KUKA KRL program: EPS_2_25862_MH08_A_20251016035158.src

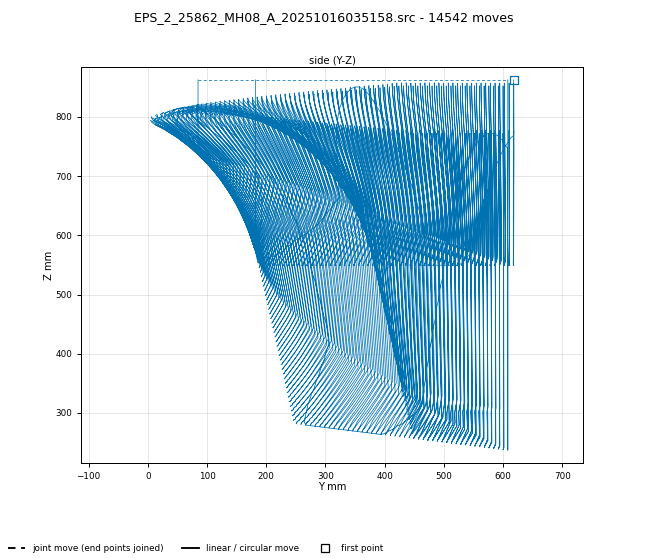
[picture p0: tool path of EPS_2_25862_MH08_A_20251016035158.src, 14542 of 14544 moves have a stored position in this frame; points joined in program order, loops and branches not executed]
&ACCESS RVP
&REL 4
&COMMENT QRS 19112012
&PARAM EDITMASK = *
DEF PART()
EXT BAS (BAS_COMMAND :IN,REAL :IN )
INT I
BAS (#INITMOV,0 )

;KUKA QRS Post kuka4.cps  Date:22-06-2017 !

File_ID=2888

QRS_PRE_INIT()

;Init var - Until changes are made in qrs_pre_init
Outlet_Square_prg=0
Inlet_1_Square_prg=0
Inlet_2_Square_prg=0
Inlet_3_Square_prg=0
Inlet_4_Square_prg=0
Inlet_5_Square_prg=0

Outlet_1={X 0.000, Y 425.000, Z 586.000, B 0.000, E1 0.000 }
Inlet_1={X 0.000, Y 425.000, Z 506.000, B 0.000, E1 105.000 }
Outlet_1_type=533
Inlet_1_type=533
;QRS#1=Sidecore dimensions
;QRS#2=525-21" Concrete
;QRS#3=525-21" Concrete
;QRS#4=
;QRS#5=
;QRS#6=
;QRS#7=
;QRS#8=
;QRS#9=S306-32
;QRS#10=S306-32
;QRS#11=
;QRS#12=
;QRS#13=
;QRS#14=
;QRS#15=
;QRS#16=1220x127x1219 4'
;QRS#17=EPS Height
;QRS#18=852,5
;QRS#19=*
;QRS#20= UPDATED VERSION 22-06-2017
;QRS#21=*
Outlet_Square=0250
Inlet_1_Square=0250
Inlet_2_Square=0
Inlet_3_Square=0
Inlet_4_Square=0
Inlet_5_Square=0
Mill_Square=1
Outlet_Square_Prg=263
Inlet_1_Square_prg=263

QRS_INIT()

$ADVANCE=5

; T1
PTP {E1 171.076,E2 171.076}
PTP {X 0,Y 617.86,A -85,B 0,C 180,E1 171.076,E2 171.076,E3 0,E4 0,E5 0,E6 0}
QRS_SPEED_INIT()
LIN {X 0,Y 617.86,Z 862.5,A -85,B 0,C 180,E1 171.076,E2 171.076,E3 0,E4 0,E5 0,E6 0} C_VEL
LIN {X 0,Y 617.86,Z 779.647,A -85,B 0,C 180,E1 171.076,E2 171.076} C_VEL
LIN {X 0,Y 617.86,Z 770.782,A -85,B 0,C 180,E1 171.076,E2 171.076} C_VEL
LIN {X 0,Y 617.855,Z 768.843,A -85,B 0,C 180,E1 171.216,E2 171.216} C_VEL
LIN {X 0,Y 617.946,Z 765.76,A -85,B 0,C 180,E1 172.353,E2 172.353} C_VEL
LIN {X 0,Y 617.789,Z 761.298,A -85,B 0,C 180,E1 173.748,E2 173.748} C_VEL
LIN {X 0,Y 617.856,Z 757.801,A -85,B 0,C 180,E1 174.678,E2 174.678} C_VEL
LIN {X 0,Y 618.003,Z 753.871,A -85,B 0,C 180,E1 175.607,E2 175.607} C_VEL
LIN {X 0,Y 617.888,Z 750.793,A -85,B 0,C 180,E1 176.301,E2 176.301} C_VEL
LIN {X 0,Y 617.795,Z 745.083,A -85,B 0,C 180,E1 177.458,E2 177.458} C_VEL
LIN {X 0,Y 617.882,Z 740.033,A -85,B 0,C 180,E1 178.384,E2 178.384} C_VEL
LIN {X 0,Y 617.968,Z 734.443,A -85,B 0,C 180,E1 179.308,E2 179.308} C_VEL
LIN {X 0,Y 617.83,Z 725.303,A -85,B 0,C 180,E1 180.695,E2 180.695} C_VEL
LIN {X 0,Y 617.888,Z 718.536,A -85,B 0,C 180,E1 181.619,E2 181.619} C_VEL
LIN {X 0,Y 617.931,Z 709.192,A -85,B 0,C 180,E1 182.776,E2 182.776} C_VEL
LIN {X 0,Y 617.867,Z 701.077,A -85,B 0,C 180,E1 183.702,E2 183.702} C_VEL
LIN {X 0,Y 617.921,Z 692.2,A -85,B 0,C 180,E1 184.628,E2 184.628} C_VEL
LIN {X 0,Y 617.95,Z 682.514,A -85,B 0,C 180,E1 185.556,E2 185.556} C_VEL
LIN {X 0,Y 617.899,Z 673.337,A -85,B 0,C 180,E1 186.37,E2 186.37} C_VEL
LIN {X 0,Y 617.909,Z 663.341,A -85,B 0,C 180,E1 187.184,E2 187.184} C_VEL
LIN {X 0,Y 617.892,Z 652.417,A -85,B 0,C 180,E1 188,E2 188} C_VEL
LIN {X 0,Y 617.911,Z 641.615,A -85,B 0,C 180,E1 188.738,E2 188.738} C_VEL
LIN {X 0,Y 617.886,Z 630.772,A -85,B 0,C 180,E1 189.418,E2 189.418} C_VEL
LIN {X 0,Y 617.869,Z 619.117,A -85,B 0,C 180,E1 190.08,E2 190.08} C_VEL
LIN {X 0,Y 617.915,Z 605.805,A -85,B 0,C 180,E1 190.752,E2 190.752} C_VEL
LIN {X 0,Y 617.872,Z 594.523,A -85,B 0,C 180,E1 191.268,E2 191.268} C_VEL
LIN {X 0,Y 617.78,Z 582.771,A -85,B 0,C 180,E1 191.749,E2 191.749} C_VEL
LIN {X 0,Y 617.848,Z 567.515,A -85,B 0,C 180,E1 192.274,E2 192.274} C_VEL
LIN {X 0,Y 617.736,Z 554.731,A -85,B 0,C 180,E1 192.655,E2 192.655} C_VEL
LIN {X 0,Y 617.593,Z 549.754,A -85,B 0,C 180,E1 192.788,E2 192.788} C_VEL
LIN {X 0,Y 617.736,Z 549.53,A -85,B 0,C 180,E1 192.822,E2 192.822} C_VEL
LIN {X 0,Y 618.063,Z 549.53,A -85,B 0,C 180,E1 192.963,E2 192.963} C_VEL
LIN {X 0,Y 617.964,Z 549.53,A -85,B 0,C 180,E1 195.199,E2 195.199} C_VEL
LIN {X 0,Y 617.909,Z 549.53,A -85,B 0,C 180,E1 200.051,E2 200.051} C_VEL
LIN {X 0,Y 617.429,Z 549.53,A -85,B 0,C 180,E1 202.55,E2 202.55} C_VEL
LIN {X 0,Y 617.883,Z 549.53,A -85,B 0,C 180,E1 205.058,E2 205.058} C_VEL
LIN {X 0,Y 617.396,Z 549.53,A -85,B 0,C 180,E1 207.661,E2 207.661} C_VEL
LIN {X 0,Y 617.869,Z 549.53,A -85,B 0,C 180,E1 210.28,E2 210.28} C_VEL
LIN {X 0,Y 617.313,Z 549.53,A -85,B 0,C 180,E1 213.028,E2 213.028} C_VEL
LIN {X 0,Y 617.774,Z 549.53,A -85,B 0,C 180,E1 215.802,E2 215.802} C_VEL
LIN {X 0,Y 617.556,Z 549.53,A -85,B 0,C 180,E1 218.097,E2 218.097} C_VEL
LIN {X 0,Y 617.539,Z 549.53,A -85,B 0,C 180,E1 218.724,E2 218.724} C_VEL
LIN {X 0,Y 617.773,Z 549.53,A -85,B 0,C 180,E1 221.734,E2 221.734} C_VEL
LIN {X 0,Y 617.845,Z 549.53,A -85,B 0,C 180,E1 225.096,E2 225.096} C_VEL
LIN {X 0,Y 617.433,Z 549.53,A -85,B 0,C 180,E1 228.311,E2 228.311} C_VEL
LIN {X 0,Y 617.775,Z 549.53,A -85,B 0,C 180,E1 231.294,E2 231.294} C_VEL
LIN {X 0,Y 617.721,Z 549.53,A -85,B 0,C 180,E1 235.803,E2 235.803} C_VEL
LIN {X 0,Y 617.906,Z 549.53,A -85,B 0,C 180,E1 237.008,E2 237.008} C_VEL
LIN {X 0,Y 618.058,Z 549.53,A -85,B 0,C 180,E1 240.653,E2 240.653} C_VEL
LIN {X 0,Y 617.765,Z 549.53,A -85,B 0,C 180,E1 240.802,E2 240.802} C_VEL
LIN {X 0,Y 617.424,Z 549.53,A -85,B 0,C 180,E1 240.866,E2 240.866} C_VEL
LIN {X 0,Y 617.177,Z 552.007,A -85,B 0,C 180,E1 240.934,E2 240.934} C_VEL
LIN {X 0,Y 617.712,Z 600.072,A -85,B 0,C 180,E1 241.593,E2 241.593} C_VEL
LIN {X 0,Y 617.671,Z 613,A -85,B 0,C 180,E1 241.802,E2 241.802} C_VEL
LIN {X 0,Y 617.749,Z 625.862,A -85,B 0,C 180,E1 242.077,E2 242.077} C_VEL
LIN {X 0,Y 617.69,Z 639.633,A -85,B 0,C 180,E1 242.435,E2 242.435} C_VEL
LIN {X 0,Y 617.845,Z 652.624,A -85,B 0,C 180,E1 242.849,E2 242.849} C_VEL
LIN {X 0,Y 617.868,Z 663.92,A -85,B 0,C 180,E1 243.255,E2 243.255} C_VEL
LIN {X 0,Y 617.757,Z 677.549,A -85,B 0,C 180,E1 243.815,E2 243.815} C_VEL
LIN {X 0,Y 617.88,Z 689.57,A -85,B 0,C 180,E1 244.383,E2 244.383} C_VEL
LIN {X 0,Y 617.885,Z 701.766,A -85,B 0,C 180,E1 245.021,E2 245.021} C_VEL
LIN {X 0,Y 617.847,Z 713.431,A -85,B 0,C 180,E1 245.696,E2 245.696} C_VEL
LIN {X 0,Y 617.909,Z 724.148,A -85,B 0,C 180,E1 246.381,E2 246.381} C_VEL
LIN {X 0,Y 617.926,Z 735.395,A -85,B 0,C 180,E1 247.169,E2 247.169} C_VEL
LIN {X 0,Y 617.917,Z 745.495,A -85,B 0,C 180,E1 247.938,E2 247.938} C_VEL
LIN {X 0,Y 617.886,Z 756.638,A -85,B 0,C 180,E1 248.868,E2 248.868} C_VEL
LIN {X 0,Y 617.923,Z 766.758,A -85,B 0,C 180,E1 249.796,E2 249.796} C_VEL
LIN {X 0,Y 617.933,Z 775.516,A -85,B 0,C 180,E1 250.667,E2 250.667} C_VEL
LIN {X 0,Y 617.881,Z 782.645,A -85,B 0,C 180,E1 251.423,E2 251.423} C_VEL
LIN {X 0,Y 617.901,Z 791.01,A -85,B 0,C 180,E1 252.391,E2 252.391} C_VEL
LIN {X 0,Y 617.982,Z 799.194,A -85,B 0,C 180,E1 253.428,E2 253.428} C_VEL
LIN {X 0,Y 617.836,Z 807.707,A -85,B 0,C 180,E1 254.61,E2 254.61} C_VEL
LIN {X 0,Y 617.888,Z 814.764,A -85,B 0,C 180,E1 255.696,E2 255.696} C_VEL
LIN {X 0,Y 617.959,Z 820.117,A -85,B 0,C 180,E1 256.59,E2 256.59} C_VEL
LIN {X 0,Y 617.783,Z 826.559,A -85,B 0,C 180,E1 257.772,E2 257.772} C_VEL
LIN {X 0,Y 617.807,Z 832.241,A -85,B 0,C 180,E1 258.952,E2 258.952} C_VEL
LIN {X 0,Y 617.978,Z 836.454,A -85,B 0,C 180,E1 259.948,E2 259.948} C_VEL
LIN {X 0,Y 617.803,Z 841.451,A -85,B 0,C 180,E1 261.248,E2 261.248} C_VEL
LIN {X 0,Y 617.803,Z 845.014,A -85,B 0,C 180,E1 262.349,E2 262.349} C_VEL
LIN {X 0,Y 617.954,Z 848.839,A -85,B 0,C 180,E1 263.748,E2 263.748} C_VEL
LIN {X 0,Y 617.79,Z 850.923,A -85,B 0,C 180,E1 264.675,E2 264.675} C_VEL
LIN {X 0,Y 617.737,Z 852.676,A -85,B 0,C 180,E1 265.603,E2 265.603} C_VEL
LIN {X 0,Y 617.832,Z 854.095,A -85,B 0,C 180,E1 266.53,E2 266.53} C_VEL
LIN {X 0,Y 617.873,Z 855.552,A -85,B 0,C 180,E1 267.919,E2 267.919} C_VEL
LIN {X 0,Y 617.747,Z 856.216,A -85,B 0,C 180,E1 268.843,E2 268.843} C_VEL
LIN {X 0,Y 617.993,Z 856.15,A -85,B 0,C 180,E1 271.154,E2 271.154} C_VEL
LIN {X 0,Y 617.755,Z 855.227,A -85,B 0,C 180,E1 272.542,E2 272.542} C_VEL
LIN {X 0,Y 617.805,Z 853.446,A -85,B 0,C 180,E1 273.931,E2 273.931} C_VEL
LIN {X 0,Y 617.985,Z 851.841,A -85,B 0,C 180,E1 274.857,E2 274.857} C_VEL
LIN {X 0,Y 617.799,Z 848.883,A -85,B 0,C 180,E1 276.252,E2 276.252} C_VEL
LIN {X 0,Y 617.849,Z 845.01,A -85,B 0,C 180,E1 277.649,E2 277.649} C_VEL
LIN {X 0,Y 617.932,Z 841.121,A -85,B 0,C 180,E1 278.829,E2 278.829} C_VEL
LIN {X 0,Y 617.775,Z 836.418,A -85,B 0,C 180,E1 280.074,E2 280.074} C_VEL
LIN {X 0,Y 617.826,Z 832.246,A -85,B 0,C 180,E1 281.046,E2 281.046} C_VEL
LIN {X 0,Y 617.969,Z 826.531,A -85,B 0,C 180,E1 282.223,E2 282.223} C_VEL
LIN {X 0,Y 617.83,Z 820.153,A -85,B 0,C 180,E1 283.411,E2 283.411} C_VEL
LIN {X 0,Y 617.902,Z 811.94,A -85,B 0,C 180,E1 284.749,E2 284.749} C_VEL
LIN {X 0,Y 617.938,Z 805.139,A -85,B 0,C 180,E1 285.757,E2 285.757} C_VEL
LIN {X 0,Y 617.865,Z 798.325,A -85,B 0,C 180,E1 286.692,E2 286.692} C_VEL
LIN {X 0,Y 617.91,Z 789.911,A -85,B 0,C 180,E1 287.739,E2 287.739} C_VEL
LIN {X 0,Y 617.968,Z 781.822,A -85,B 0,C 180,E1 288.664,E2 288.664} C_VEL
LIN {X 0,Y 617.898,Z 771.912,A -85,B 0,C 180,E1 289.702,E2 289.702} C_VEL
LIN {X 0,Y 617.915,Z 763.54,A -85,B 0,C 180,E1 290.51,E2 290.51} C_VEL
LIN {X 0,Y 617.932,Z 753.044,A -85,B 0,C 180,E1 291.438,E2 291.438} C_VEL
LIN {X 0,Y 617.906,Z 743.508,A -85,B 0,C 180,E1 292.217,E2 292.217} C_VEL
LIN {X 0,Y 617.904,Z 733.665,A -85,B 0,C 180,E1 292.958,E2 292.958} C_VEL
LIN {X 0,Y 617.855,Z 722.1,A -85,B 0,C 180,E1 293.755,E2 293.755} C_VEL
LIN {X 0,Y 617.9,Z 709.896,A -85,B 0,C 180,E1 294.512,E2 294.512} C_VEL
LIN {X 0,Y 617.869,Z 698.904,A -85,B 0,C 180,E1 295.136,E2 295.136} C_VEL
LIN {X 0,Y 617.811,Z 688.04,A -85,B 0,C 180,E1 295.698,E2 295.698} C_VEL
LIN {X 0,Y 617.891,Z 673.891,A -85,B 0,C 180,E1 296.338,E2 296.338} C_VEL
LIN {X 0,Y 617.852,Z 660.692,A -85,B 0,C 180,E1 296.865,E2 296.865} C_VEL
LIN {X 0,Y 617.731,Z 650.39,A -85,B 0,C 180,E1 297.235,E2 297.235} C_VEL
LIN {X 0,Y 617.857,Z 634.553,A -85,B 0,C 180,E1 297.698,E2 297.698} C_VEL
LIN {X 0,Y 617.754,Z 621.8,A -85,B 0,C 180,E1 298.016,E2 298.016} C_VEL
LIN {X 0,Y 617.683,Z 612.51,A -85,B 0,C 180,E1 298.208,E2 298.208} C_VEL
LIN {X 0,Y 617.674,Z 593.335,A -85,B 0,C 180,E1 298.503,E2 298.503} C_VEL
LIN {X 0,Y 617.203,Z 549.53,A -85,B 0,C 180,E1 299.103,E2 299.103} C_VEL
LIN {X 0,Y 618.035,Z 549.53,A -85,B 0,C 180,E1 299.981,E2 299.981} C_VEL
LIN {X 0,Y 618.046,Z 549.53,A -85,B 0,C 180,E1 300.268,E2 300.268} C_VEL
LIN {X 0,Y 617.365,Z 549.53,A -85,B 0,C 180,E1 304.149,E2 304.149} C_VEL
LIN {X 0,Y 617.816,Z 549.53,A -85,B 0,C 180,E1 305.796,E2 305.796} C_VEL
LIN {X 0,Y 617.559,Z 549.53,A -85,B 0,C 180,E1 308.719,E2 308.719} C_VEL
LIN {X 0,Y 617.784,Z 549.53,A -85,B 0,C 180,E1 311.73,E2 311.73} C_VEL
LIN {X 0,Y 617.826,Z 549.53,A -85,B 0,C 180,E1 315.094,E2 315.094} C_VEL
LIN {X 0,Y 617.429,Z 549.53,A -85,B 0,C 180,E1 318.308,E2 318.308} C_VEL
LIN {X 0,Y 617.778,Z 549.53,A -85,B 0,C 180,E1 321.294,E2 321.294} C_VEL
LIN {X 0,Y 617.698,Z 549.53,A -85,B 0,C 180,E1 325.802,E2 325.802} C_VEL
LIN {X 0,Y 617.852,Z 549.53,A -85,B 0,C 180,E1 327.005,E2 327.005} C_VEL
LIN {X 0,Y 617.635,Z 549.53,A -85,B 0,C 180,E1 330.173,E2 330.173} C_VEL
LIN {X 0,Y 617.65,Z 549.53,A -85,B 0,C 180,E1 332.351,E2 332.351} C_VEL
LIN {X 0,Y 617.511,Z 549.53,A -85,B 0,C 180,E1 335.24,E2 335.24} C_VEL
LIN {X 0,Y 617.715,Z 549.53,A -85,B 0,C 180,E1 337.461,E2 337.461} C_VEL
LIN {X 0,Y 617.711,Z 549.53,A -85,B 0,C 180,E1 341.463,E2 341.463} C_VEL
LIN {X 0,Y 617.916,Z 549.53,A -85,B 0,C 180,E1 342.391,E2 342.391} C_VEL
LIN {X 0,Y 617.972,Z 549.53,A -85,B 0,C 180,E1 347.183,E2 347.183} C_VEL
LIN {X 0,Y 617.993,Z 549.53,A -85,B 0,C 180,E1 351.884,E2 351.884} C_VEL
LIN {X 0,Y 617.983,Z 549.53,A -85,B 0,C 180,E1 356.53,E2 356.53} C_VEL
LIN {X 0,Y 618.035,Z 549.53,A -85,B 0,C 180,E1 361.154,E2 361.154} C_VEL
LIN {X 0,Y 618.003,Z 549.53,A -85,B 0,C 180,E1 365.785,E2 365.785} C_VEL
LIN {X 0,Y 617.942,Z 549.53,A -85,B 0,C 180,E1 370.455,E2 370.455} C_VEL
LIN {X 0,Y 617.951,Z 549.53,A -85,B 0,C 180,E1 375.196,E2 375.196} C_VEL
LIN {X 0,Y 617.911,Z 549.53,A -85,B 0,C 180,E1 380.048,E2 380.048} C_VEL
LIN {X 0,Y 617.428,Z 549.53,A -85,B 0,C 180,E1 382.547,E2 382.547} C_VEL
LIN {X 0,Y 617.88,Z 549.53,A -85,B 0,C 180,E1 385.055,E2 385.055} C_VEL
LIN {X 0,Y 617.373,Z 549.53,A -85,B 0,C 180,E1 387.659,E2 387.659} C_VEL
LIN {X 0,Y 617.823,Z 549.53,A -85,B 0,C 180,E1 390.279,E2 390.279} C_VEL
LIN {X 0,Y 617.307,Z 549.53,A -85,B 0,C 180,E1 393.025,E2 393.025} C_VEL
LIN {X 0,Y 617.797,Z 549.53,A -85,B 0,C 180,E1 395.797,E2 395.797} C_VEL
LIN {X 0,Y 617.55,Z 549.53,A -85,B 0,C 180,E1 398.1,E2 398.1} C_VEL
LIN {X 0,Y 617.522,Z 549.53,A -85,B 0,C 180,E1 398.721,E2 398.721} C_VEL
LIN {X 0,Y 617.73,Z 549.53,A -85,B 0,C 180,E1 401.733,E2 401.733} C_VEL
LIN {X 0,Y 617.827,Z 549.53,A -85,B 0,C 180,E1 405.097,E2 405.097} C_VEL
LIN {X 0,Y 617.414,Z 549.53,A -85,B 0,C 180,E1 408.308,E2 408.308} C_VEL
LIN {X 0,Y 617.756,Z 549.53,A -85,B 0,C 180,E1 411.295,E2 411.295} C_VEL
LIN {X 0,Y 617.695,Z 549.53,A -85,B 0,C 180,E1 415.801,E2 415.801} C_VEL
LIN {X 0,Y 617.863,Z 549.53,A -85,B 0,C 180,E1 417.008,E2 417.008} C_VEL
LIN {X 0,Y 617.607,Z 549.53,A -85,B 0,C 180,E1 420.176,E2 420.176} C_VEL
LIN {X 0,Y 617.623,Z 549.53,A -85,B 0,C 180,E1 422.352,E2 422.352} C_VEL
LIN {X 0,Y 617.494,Z 549.53,A -85,B 0,C 180,E1 425.241,E2 425.241} C_VEL
LIN {X 0,Y 617.726,Z 549.53,A -85,B 0,C 180,E1 427.464,E2 427.464} C_VEL
LIN {X 0,Y 617.74,Z 549.53,A -85,B 0,C 180,E1 431.452,E2 431.452} C_VEL
LIN {X 0,Y 617.966,Z 549.53,A -85,B 0,C 180,E1 432.395,E2 432.395} C_VEL
LIN {X 0,Y 617.987,Z 549.53,A -85,B 0,C 180,E1 437.186,E2 437.186} C_VEL
LIN {X 0,Y 617.989,Z 549.53,A -85,B 0,C 180,E1 441.887,E2 441.887} C_VEL
LIN {X 0,Y 618.059,Z 549.53,A -85,B 0,C 180,E1 446.533,E2 446.533} C_VEL
LIN {X 0,Y 618.057,Z 549.53,A -85,B 0,C 180,E1 451.156,E2 451.156} C_VEL
LIN {X 0,Y 618,Z 549.53,A -85,B 0,C 180,E1 455.787,E2 455.787} C_VEL
LIN {X 0,Y 617.992,Z 549.53,A -85,B 0,C 180,E1 460.457,E2 460.457} C_VEL
LIN {X 0,Y 617.977,Z 549.53,A -85,B 0,C 180,E1 465.198,E2 465.198} C_VEL
LIN {X 0,Y 617.929,Z 549.53,A -85,B 0,C 180,E1 470.05,E2 470.05} C_VEL
LIN {X 0,Y 617.46,Z 549.53,A -85,B 0,C 180,E1 472.548,E2 472.548} C_VEL
LIN {X 0,Y 617.927,Z 549.53,A -85,B 0,C 180,E1 475.056,E2 475.056} C_VEL
LIN {X 0,Y 617.423,Z 549.53,A -85,B 0,C 180,E1 477.66,E2 477.66} C_VEL
LIN {X 0,Y 617.873,Z 549.53,A -85,B 0,C 180,E1 480.279,E2 480.279} C_VEL
LIN {X 0,Y 617.335,Z 549.53,A -85,B 0,C 180,E1 483.026,E2 483.026} C_VEL
LIN {X 0,Y 617.801,Z 549.53,A -85,B 0,C 180,E1 485.8,E2 485.8} C_VEL
LIN {X 0,Y 617.577,Z 549.53,A -85,B 0,C 180,E1 488.104,E2 488.104} C_VEL
LIN {X 0,Y 617.55,Z 549.53,A -85,B 0,C 180,E1 488.722,E2 488.722} C_VEL
LIN {X 0,Y 617.688,Z 549.53,A -85,B 0,C 180,E1 491.74,E2 491.74} C_VEL
LIN {X 0,Y 617.79,Z 549.53,A -85,B 0,C 180,E1 496.317,E2 496.317} C_VEL
LIN {X 0,Y 617.839,Z 549.53,A -85,B 0,C 180,E1 497.021,E2 497.021} C_VEL
LIN {X 0,Y 617.397,Z 549.568,A -85,B 0,C 180,E1 497.108,E2 497.108} C_VEL
LIN {X 0,Y 617.63,Z 560.15,A -85,B 0,C 180,E1 497.403,E2 497.403} C_VEL
LIN {X 0,Y 617.807,Z 572.726,A -85,B 0,C 180,E1 497.806,E2 497.806} C_VEL
LIN {X 0,Y 617.864,Z 585.591,A -85,B 0,C 180,E1 498.278,E2 498.278} C_VEL
LIN {X 0,Y 617.802,Z 596.785,A -85,B 0,C 180,E1 498.737,E2 498.737} C_VEL
LIN {X 0,Y 617.893,Z 610.519,A -85,B 0,C 180,E1 499.387,E2 499.387} C_VEL
LIN {X 0,Y 617.909,Z 621.273,A -85,B 0,C 180,E1 499.949,E2 499.949} C_VEL
LIN {X 0,Y 617.883,Z 633.063,A -85,B 0,C 180,E1 500.63,E2 500.63} C_VEL
LIN {X 0,Y 617.896,Z 645.621,A -85,B 0,C 180,E1 501.438,E2 501.438} C_VEL
LIN {X 0,Y 617.909,Z 656.566,A -85,B 0,C 180,E1 502.212,E2 502.212} C_VEL
LIN {X 0,Y 617.926,Z 667.227,A -85,B 0,C 180,E1 503.036,E2 503.036} C_VEL
LIN {X 0,Y 617.9,Z 677.544,A -85,B 0,C 180,E1 503.906,E2 503.906} C_VEL
LIN {X 0,Y 617.865,Z 685.157,A -85,B 0,C 180,E1 504.592,E2 504.592} C_VEL
LIN {X 0,Y 617.918,Z 694.828,A -85,B 0,C 180,E1 505.548,E2 505.548} C_VEL
LIN {X 0,Y 617.931,Z 704.001,A -85,B 0,C 180,E1 506.537,E2 506.537} C_VEL
LIN {X 0,Y 617.851,Z 711.454,A -85,B 0,C 180,E1 507.4,E2 507.4} C_VEL
LIN {X 0,Y 617.895,Z 720.414,A -85,B 0,C 180,E1 508.547,E2 508.547} C_VEL
LIN {X 0,Y 617.953,Z 727.645,A -85,B 0,C 180,E1 509.561,E2 509.561} C_VEL
LIN {X 0,Y 617.826,Z 734.192,A -85,B 0,C 180,E1 510.552,E2 510.552} C_VEL
LIN {X 0,Y 617.836,Z 739.902,A -85,B 0,C 180,E1 511.502,E2 511.502} C_VEL
LIN {X 0,Y 617.978,Z 746.346,A -85,B 0,C 180,E1 512.696,E2 512.696} C_VEL
LIN {X 0,Y 617.79,Z 752.56,A -85,B 0,C 180,E1 513.98,E2 513.98} C_VEL
LIN {X 0,Y 617.811,Z 757.639,A -85,B 0,C 180,E1 515.184,E2 515.184} C_VEL
LIN {X 0,Y 617.969,Z 761.298,A -85,B 0,C 180,E1 516.175,E2 516.175} C_VEL
LIN {X 0,Y 617.771,Z 765.547,A -85,B 0,C 180,E1 517.467,E2 517.467} C_VEL
LIN {X 0,Y 617.759,Z 768.917,A -85,B 0,C 180,E1 518.712,E2 518.712} C_VEL
LIN {X 0,Y 617.967,Z 771.586,A -85,B 0,C 180,E1 519.954,E2 519.954} C_VEL
LIN {X 0,Y 617.768,Z 774.076,A -85,B 0,C 180,E1 521.454,E2 521.454} C_VEL
LIN {X 0,Y 617.781,Z 775.193,A -85,B 0,C 180,E1 522.39,E2 522.39} C_VEL
LIN {X 0,Y 617.978,Z 776.052,A -85,B 0,C 180,E1 523.609,E2 523.609} C_VEL
LIN {X 0,Y 617.929,Z 776.402,A -85,B 0,C 180,E1 524.804,E2 524.804} C_VEL
LIN {X 0,Y 617.975,Z 776.178,A -85,B 0,C 180,E1 525.999,E2 525.999} C_VEL
LIN {X 0,Y 617.892,Z 775.444,A -85,B 0,C 180,E1 527.185,E2 527.185} C_VEL
LIN {X 0,Y 617.968,Z 774.124,A -85,B 0,C 180,E1 528.368,E2 528.368} C_VEL
LIN {X 0,Y 617.83,Z 772.331,A -85,B 0,C 180,E1 529.543,E2 529.543} C_VEL
LIN {X 0,Y 617.778,Z 770.792,A -85,B 0,C 180,E1 530.341,E2 530.341} C_VEL
LIN {X 0,Y 617.855,Z 768.843,A -85,B 0,C 180,E1 531.216,E2 531.216} C_VEL
LIN {X 0,Y 613.894,Z 765.328,A -85,B 0,C 180,E1 532.764,E2 532.764} C_VEL
LIN {X 0,Y 610.005,Z 760.35,A -85,B 0,C 180,E1 534.311,E2 534.311} C_VEL
LIN {X 0,Y 609.99,Z 746.173,A -85,B 0,C 180,E1 537.508,E2 537.508} C_VEL
LIN {X 0,Y 610.077,Z 725.651,A -85,B 0,C 180,E1 540.886,E2 540.886} C_VEL
LIN {X 0,Y 610.19,Z 699.825,A -85,B 0,C 180,E1 544.088,E2 544.088} C_VEL
LIN {X 0,Y 610.347,Z 669.143,A -85,B 0,C 180,E1 547,E2 547} C_VEL
LIN {X 0,Y 610.508,Z 635.253,A -85,B 0,C 180,E1 549.453,E2 549.453} C_VEL
LIN {X 0,Y 610.693,Z 598.195,A -85,B 0,C 180,E1 551.437,E2 551.437} C_VEL
LIN {X 0,Y 610.749,Z 560.222,A -85,B 0,C 180,E1 552.843,E2 552.843} C_VEL
LIN {X 0,Y 610.127,Z 549.53,A -85,B 0,C 180,E1 553.176,E2 553.176} C_VEL
LIN {X 0,Y 609.735,Z 549.53,A -85,B 0,C 180,E1 559.333,E2 559.333} C_VEL
LIN {X 0,Y 609.966,Z 549.53,A -85,B 0,C 180,E1 564.955,E2 564.955} C_VEL
LIN {X 0,Y 609.791,Z 549.53,A -85,B 0,C 180,E1 569.77,E2 569.77} C_VEL
LIN {X 0,Y 609.693,Z 549.53,A -85,B 0,C 180,E1 576.579,E2 576.579} C_VEL
LIN {X 0,Y 609.779,Z 549.53,A -85,B 0,C 180,E1 582.093,E2 582.093} C_VEL
LIN {X 0,Y 609.475,Z 549.53,A -85,B 0,C 180,E1 587.875,E2 587.875} C_VEL
LIN {X 0,Y 609.473,Z 549.53,A -85,B 0,C 180,E1 592.644,E2 592.644} C_VEL
LIN {X 0,Y 609.892,Z 549.53,A -85,B 0,C 180,E1 597.563,E2 597.563} C_VEL
LIN {X 0,Y 610.106,Z 549.53,A -85,B 0,C 180,E1 600.523,E2 600.523} C_VEL
LIN {X 0,Y 610.754,Z 622.437,A -85,B 0,C 180,E1 601.647,E2 601.647} C_VEL
LIN {X 0,Y 610.743,Z 662.256,A -85,B 0,C 180,E1 602.853,E2 602.853} C_VEL
LIN {X 0,Y 610.622,Z 699.55,A -85,B 0,C 180,E1 604.578,E2 604.578} C_VEL
LIN {X 0,Y 610.442,Z 735.861,A -85,B 0,C 180,E1 606.908,E2 606.908} C_VEL
LIN {X 0,Y 610.29,Z 768.229,A -85,B 0,C 180,E1 609.676,E2 609.676} C_VEL
LIN {X 0,Y 610.174,Z 795.223,A -85,B 0,C 180,E1 612.676,E2 612.676} C_VEL
LIN {X 0,Y 610.125,Z 818.057,A -85,B 0,C 180,E1 615.998,E2 615.998} C_VEL
LIN {X 0,Y 610.106,Z 836.363,A -85,B 0,C 180,E1 619.634,E2 619.634} C_VEL
LIN {X 0,Y 610.02,Z 848.178,A -85,B 0,C 180,E1 623.081,E2 623.081} C_VEL
LIN {X 0,Y 609.912,Z 853.931,A -85,B 0,C 180,E1 625.728,E2 625.728} C_VEL
LIN {X 0,Y 609.965,Z 857.082,A -85,B 0,C 180,E1 628.577,E2 628.577} C_VEL
LIN {X 0,Y 610.111,Z 857.083,A -85,B 0,C 180,E1 631.421,E2 631.421} C_VEL
LIN {X 0,Y 610.17,Z 852.727,A -85,B 0,C 180,E1 634.982,E2 634.982} C_VEL
LIN {X 0,Y 610.108,Z 841.962,A -85,B 0,C 180,E1 638.922,E2 638.922} C_VEL
LIN {X 0,Y 610.133,Z 826.223,A -85,B 0,C 180,E1 642.54,E2 642.54} C_VEL
LIN {X 0,Y 610.147,Z 804.955,A -85,B 0,C 180,E1 646.025,E2 646.025} C_VEL
LIN {X 0,Y 610.251,Z 778.826,A -85,B 0,C 180,E1 649.237,E2 649.237} C_VEL
LIN {X 0,Y 610.37,Z 749.245,A -85,B 0,C 180,E1 652.035,E2 652.035} C_VEL
LIN {X 0,Y 610.509,Z 715.147,A -85,B 0,C 180,E1 654.505,E2 654.505} C_VEL
LIN {X 0,Y 610.67,Z 678.777,A -85,B 0,C 180,E1 656.455,E2 656.455} C_VEL
LIN {X 0,Y 610.792,Z 641.071,A -85,B 0,C 180,E1 657.859,E2 657.859} C_VEL
LIN {X 0,Y 610.76,Z 603.673,A -85,B 0,C 180,E1 658.704,E2 658.704} C_VEL
LIN {X 0,Y 609.662,Z 549.53,A -85,B 0,C 180,E1 659.499,E2 659.499} C_VEL
LIN {X 0,Y 609.635,Z 549.53,A -85,B 0,C 180,E1 664.965,E2 664.965} C_VEL
LIN {X 0,Y 609.573,Z 549.53,A -85,B 0,C 180,E1 670.224,E2 670.224} C_VEL
LIN {X 0,Y 609.703,Z 549.53,A -85,B 0,C 180,E1 674.052,E2 674.052} C_VEL
LIN {X 0,Y 609.602,Z 549.53,A -85,B 0,C 180,E1 680.348,E2 680.348} C_VEL
LIN {X 0,Y 609.928,Z 549.53,A -85,B 0,C 180,E1 686.903,E2 686.903} C_VEL
LIN {X 0,Y 609.685,Z 549.53,A -85,B 0,C 180,E1 691.851,E2 691.851} C_VEL
LIN {X 0,Y 609.65,Z 549.53,A -85,B 0,C 180,E1 696.763,E2 696.763} C_VEL
LIN {X 0,Y 609.915,Z 549.53,A -85,B 0,C 180,E1 702.673,E2 702.673} C_VEL
LIN {X 0,Y 610.027,Z 549.53,A -85,B 0,C 180,E1 707.096,E2 707.096} C_VEL
LIN {X 0,Y 609.77,Z 549.53,A -85,B 0,C 180,E1 712.872,E2 712.872} C_VEL
LIN {X 0,Y 609.864,Z 549.53,A -85,B 0,C 180,E1 717.157,E2 717.157} C_VEL
LIN {X 0,Y 610.02,Z 549.53,A -85,B 0,C 180,E1 721.425,E2 721.425} C_VEL
LIN {X 0,Y 609.769,Z 549.53,A -85,B 0,C 180,E1 726.688,E2 726.688} C_VEL
LIN {X 0,Y 609.705,Z 549.53,A -85,B 0,C 180,E1 731.461,E2 731.461} C_VEL
LIN {X 0,Y 609.797,Z 549.53,A -85,B 0,C 180,E1 735.853,E2 735.853} C_VEL
LIN {X 0,Y 609.893,Z 549.53,A -85,B 0,C 180,E1 740.34,E2 740.34} C_VEL
LIN {X 0,Y 609.958,Z 549.53,A -85,B 0,C 180,E1 744.962,E2 744.962} C_VEL
LIN {X 0,Y 609.744,Z 549.53,A -85,B 0,C 180,E1 749.779,E2 749.779} C_VEL
LIN {X 0,Y 609.704,Z 549.53,A -85,B 0,C 180,E1 756.586,E2 756.586} C_VEL
LIN {X 0,Y 609.761,Z 549.53,A -85,B 0,C 180,E1 762.102,E2 762.102} C_VEL
LIN {X 0,Y 609.482,Z 549.53,A -85,B 0,C 180,E1 767.877,E2 767.877} C_VEL
LIN {X 0,Y 609.462,Z 549.53,A -85,B 0,C 180,E1 772.655,E2 772.655} C_VEL
LIN {X 0,Y 609.777,Z 549.53,A -85,B 0,C 180,E1 777.591,E2 777.591} C_VEL
LIN {X 0,Y 609.659,Z 549.53,A -85,B 0,C 180,E1 781.846,E2 781.846} C_VEL
LIN {X 0,Y 609.653,Z 549.53,A -85,B 0,C 180,E1 786.768,E2 786.768} C_VEL
LIN {X 0,Y 609.964,Z 549.53,A -85,B 0,C 180,E1 792.671,E2 792.671} C_VEL
LIN {X 0,Y 610.04,Z 549.53,A -85,B 0,C 180,E1 797.093,E2 797.093} C_VEL
LIN {X 0,Y 609.788,Z 549.53,A -85,B 0,C 180,E1 802.869,E2 802.869} C_VEL
LIN {X 0,Y 609.934,Z 549.53,A -85,B 0,C 180,E1 807.155,E2 807.155} C_VEL
LIN {X 0,Y 610.042,Z 549.53,A -85,B 0,C 180,E1 811.423,E2 811.423} C_VEL
LIN {X 0,Y 609.784,Z 549.53,A -85,B 0,C 180,E1 816.682,E2 816.682} C_VEL
LIN {X 0,Y 609.75,Z 549.53,A -85,B 0,C 180,E1 821.458,E2 821.458} C_VEL
LIN {X 0,Y 609.823,Z 549.53,A -85,B 0,C 180,E1 825.85,E2 825.85} C_VEL
LIN {X 0,Y 609.915,Z 549.53,A -85,B 0,C 180,E1 830.338,E2 830.338} C_VEL
LIN {X 0,Y 610.001,Z 549.53,A -85,B 0,C 180,E1 834.959,E2 834.959} C_VEL
LIN {X 0,Y 609.804,Z 549.53,A -85,B 0,C 180,E1 839.774,E2 839.774} C_VEL
LIN {X 0,Y 609.717,Z 549.53,A -85,B 0,C 180,E1 846.583,E2 846.583} C_VEL
LIN {X 0,Y 609.647,Z 549.53,A -85,B 0,C 180,E1 852.11,E2 852.11} C_VEL
LIN {X 0,Y 609.952,Z 550.16,A -85,B 0,C 180,E1 856.753,E2 856.753} C_VEL
LIN {X 0,Y 610.691,Z 589.728,A -85,B 0,C 180,E1 858.11,E2 858.11} C_VEL
LIN {X 0,Y 610.586,Z 625.145,A -85,B 0,C 180,E1 859.853,E2 859.853} C_VEL
LIN {X 0,Y 610.42,Z 659.882,A -85,B 0,C 180,E1 862.172,E2 862.172} C_VEL
LIN {X 0,Y 610.246,Z 691.598,A -85,B 0,C 180,E1 864.961,E2 864.961} C_VEL
LIN {X 0,Y 610.129,Z 719.48,A -85,B 0,C 180,E1 868.172,E2 868.172} C_VEL
LIN {X 0,Y 610.051,Z 742.167,A -85,B 0,C 180,E1 871.66,E2 871.66} C_VEL
LIN {X 0,Y 609.984,Z 758.264,A -85,B 0,C 180,E1 875.039,E2 875.039} C_VEL
LIN {X 0,Y 609.912,Z 768.448,A -85,B 0,C 180,E1 878.136,E2 878.136} C_VEL
LIN {X 0,Y 609.982,Z 774.752,A -85,B 0,C 180,E1 881.172,E2 881.172} C_VEL
LIN {X 0,Y 610.113,Z 777.318,A -85,B 0,C 180,E1 884.156,E2 884.156} C_VEL
LIN {X 0,Y 610.08,Z 776.575,A -85,B 0,C 180,E1 887.091,E2 887.091} C_VEL
LIN {X 0,Y 609.968,Z 771.05,A -85,B 0,C 180,E1 890.712,E2 890.712} C_VEL
LIN {X 0,Y 609.974,Z 761.731,A -85,B 0,C 180,E1 893.941,E2 893.941} C_VEL
LIN {X 0,Y 610.005,Z 760.35,A -85,B 0,C 180,E1 894.311,E2 894.311} C_VEL
LIN {X 0,Y 608.793,Z 757.49,A -85,B 0,C 180,E1 895.079,E2 895.079} C_VEL
LIN {X 0,Y 602.231,Z 748.821,A -85,B 0,C 180,E1 897.139,E2 897.139} C_VEL
LIN {X 0,Y 602.139,Z 747.912,A -85,B 0,C 180,E1 897.33,E2 897.33} C_VEL
LIN {X 0,Y 602.274,Z 727.061,A -85,B 0,C 180,E1 900.897,E2 900.897} C_VEL
LIN {X 0,Y 602.509,Z 701.685,A -85,B 0,C 180,E1 904.14,E2 904.14} C_VEL
LIN {X 0,Y 602.805,Z 671.529,A -85,B 0,C 180,E1 907.088,E2 907.088} C_VEL
LIN {X 0,Y 603.131,Z 638.374,A -85,B 0,C 180,E1 909.57,E2 909.57} C_VEL
LIN {X 0,Y 603.494,Z 602.47,A -85,B 0,C 180,E1 911.575,E2 911.575} C_VEL
LIN {X 0,Y 603.699,Z 565.232,A -85,B 0,C 180,E1 913.042,E2 913.042} C_VEL
LIN {X 0,Y 602.806,Z 552.583,A -85,B 0,C 180,E1 913.46,E2 913.46} C_VEL
LIN {X 0,Y 602.151,Z 549.53,A -85,B 0,C 180,E1 913.631,E2 913.631} C_VEL
LIN {X 0,Y 601.918,Z 549.53,A -85,B 0,C 180,E1 920.615,E2 920.615} C_VEL
LIN {X 0,Y 601.949,Z 549.53,A -85,B 0,C 180,E1 925.311,E2 925.311} C_VEL
LIN {X 0,Y 601.693,Z 549.53,A -85,B 0,C 180,E1 931.178,E2 931.178} C_VEL
LIN {X 0,Y 601.74,Z 549.53,A -85,B 0,C 180,E1 937.143,E2 937.143} C_VEL
LIN {X 0,Y 601.756,Z 549.53,A -85,B 0,C 180,E1 943.141,E2 943.141} C_VEL
LIN {X 0,Y 601.553,Z 549.53,A -85,B 0,C 180,E1 949.125,E2 949.125} C_VEL
LIN {X 0,Y 601.487,Z 549.53,A -85,B 0,C 180,E1 953.652,E2 953.652} C_VEL
LIN {X 0,Y 601.929,Z 549.53,A -85,B 0,C 180,E1 958.114,E2 958.114} C_VEL
LIN {X 0,Y 602.087,Z 549.53,A -85,B 0,C 180,E1 960.099,E2 960.099} C_VEL
LIN {X 0,Y 603.482,Z 560.306,A -85,B 0,C 180,E1 960.321,E2 960.321} C_VEL
LIN {X 0,Y 603.784,Z 624.293,A -85,B 0,C 180,E1 961.331,E2 961.331} C_VEL
LIN {X 0,Y 603.621,Z 663.138,A -85,B 0,C 180,E1 962.54,E2 962.54} C_VEL
LIN {X 0,Y 603.311,Z 701.318,A -85,B 0,C 180,E1 964.348,E2 964.348} C_VEL
LIN {X 0,Y 602.968,Z 737.346,A -85,B 0,C 180,E1 966.721,E2 966.721} C_VEL
LIN {X 0,Y 602.664,Z 768.229,A -85,B 0,C 180,E1 969.407,E2 969.407} C_VEL
LIN {X 0,Y 602.413,Z 795.224,A -85,B 0,C 180,E1 972.446,E2 972.446} C_VEL
LIN {X 0,Y 602.278,Z 818.058,A -85,B 0,C 180,E1 975.811,E2 975.811} C_VEL
LIN {X 0,Y 602.175,Z 835.446,A -85,B 0,C 180,E1 979.278,E2 979.278} C_VEL
LIN {X 0,Y 602.116,Z 847.612,A -85,B 0,C 180,E1 982.777,E2 982.777} C_VEL
LIN {X 0,Y 602.035,Z 853.931,A -85,B 0,C 180,E1 985.672,E2 985.672} C_VEL
LIN {X 0,Y 602.064,Z 857.082,A -85,B 0,C 180,E1 988.558,E2 988.558} C_VEL
LIN {X 0,Y 602.204,Z 857.083,A -85,B 0,C 180,E1 991.44,E2 991.44} C_VEL
LIN {X 0,Y 602.284,Z 852.727,A -85,B 0,C 180,E1 995.047,E2 995.047} C_VEL
LIN {X 0,Y 602.203,Z 841.963,A -85,B 0,C 180,E1 999.04,E2 999.04} C_VEL
LIN {X 0,Y 602.253,Z 826.224,A -85,B 0,C 180,E1 1002.707,E2 1002.707} C_VEL
LIN {X 0,Y 602.339,Z 805.234,A -85,B 0,C 180,E1 1006.199,E2 1006.199} C_VEL
LIN {X 0,Y 602.556,Z 779.123,A -85,B 0,C 180,E1 1009.461,E2 1009.461} C_VEL
LIN {X 0,Y 602.826,Z 749.465,A -85,B 0,C 180,E1 1012.307,E2 1012.307} C_VEL
LIN {X 0,Y 603.149,Z 716.06,A -85,B 0,C 180,E1 1014.765,E2 1014.765} C_VEL
LIN {X 0,Y 603.486,Z 679.841,A -85,B 0,C 180,E1 1016.745,E2 1016.745} C_VEL
LIN {X 0,Y 603.735,Z 643.127,A -85,B 0,C 180,E1 1018.15,E2 1018.15} C_VEL
LIN {X 0,Y 603.823,Z 606.296,A -85,B 0,C 180,E1 1019.024,E2 1019.024} C_VEL
LIN {X 0,Y 603.06,Z 553.464,A -85,B 0,C 180,E1 1019.794,E2 1019.794} C_VEL
LIN {X 0,Y 601.953,Z 549.53,A -85,B 0,C 180,E1 1019.934,E2 1019.934} C_VEL
LIN {X 0,Y 601.783,Z 549.53,A -85,B 0,C 180,E1 1026.386,E2 1026.386} C_VEL
LIN {X 0,Y 601.743,Z 549.53,A -85,B 0,C 180,E1 1030.995,E2 1030.995} C_VEL
LIN {X 0,Y 601.685,Z 549.53,A -85,B 0,C 180,E1 1035.21,E2 1035.21} C_VEL
LIN {X 0,Y 601.789,Z 549.53,A -85,B 0,C 180,E1 1041.254,E2 1041.254} C_VEL
LIN {X 0,Y 601.871,Z 549.53,A -85,B 0,C 180,E1 1046.402,E2 1046.402} C_VEL
LIN {X 0,Y 601.78,Z 549.53,A -85,B 0,C 180,E1 1051.713,E2 1051.713} C_VEL
LIN {X 0,Y 601.688,Z 549.53,A -85,B 0,C 180,E1 1056.262,E2 1056.262} C_VEL
LIN {X 0,Y 601.927,Z 549.53,A -85,B 0,C 180,E1 1062.907,E2 1062.907} C_VEL
LIN {X 0,Y 601.811,Z 549.53,A -85,B 0,C 180,E1 1068.392,E2 1068.392} C_VEL
LIN {X 0,Y 601.87,Z 549.53,A -85,B 0,C 180,E1 1072.777,E2 1072.777} C_VEL
LIN {X 0,Y 601.968,Z 549.53,A -85,B 0,C 180,E1 1077.12,E2 1077.12} C_VEL
LIN {X 0,Y 602.11,Z 549.53,A -85,B 0,C 180,E1 1081.444,E2 1081.444} C_VEL
LIN {X 0,Y 602.172,Z 549.53,A -85,B 0,C 180,E1 1085.775,E2 1085.775} C_VEL
LIN {X 0,Y 601.795,Z 549.53,A -85,B 0,C 180,E1 1091.614,E2 1091.614} C_VEL
LIN {X 0,Y 601.83,Z 549.53,A -85,B 0,C 180,E1 1096.068,E2 1096.068} C_VEL
LIN {X 0,Y 601.726,Z 549.53,A -85,B 0,C 180,E1 1101.411,E2 1101.411} C_VEL
LIN {X 0,Y 601.948,Z 549.53,A -85,B 0,C 180,E1 1105.318,E2 1105.318} C_VEL
LIN {X 0,Y 601.639,Z 549.53,A -85,B 0,C 180,E1 1111.171,E2 1111.171} C_VEL
LIN {X 0,Y 601.751,Z 549.53,A -85,B 0,C 180,E1 1117.15,E2 1117.15} C_VEL
LIN {X 0,Y 601.729,Z 549.53,A -85,B 0,C 180,E1 1123.14,E2 1123.14} C_VEL
LIN {X 0,Y 601.535,Z 549.53,A -85,B 0,C 180,E1 1129.125,E2 1129.125} C_VEL
LIN {X 0,Y 601.463,Z 549.53,A -85,B 0,C 180,E1 1133.665,E2 1133.665} C_VEL
LIN {X 0,Y 601.786,Z 549.53,A -85,B 0,C 180,E1 1138.107,E2 1138.107} C_VEL
LIN {X 0,Y 601.64,Z 549.53,A -85,B 0,C 180,E1 1143.066,E2 1143.066} C_VEL
LIN {X 0,Y 601.64,Z 549.53,A -85,B 0,C 180,E1 1148.616,E2 1148.616} C_VEL
LIN {X 0,Y 601.976,Z 549.53,A -85,B 0,C 180,E1 1152.899,E2 1152.899} C_VEL
LIN {X 0,Y 601.826,Z 549.53,A -85,B 0,C 180,E1 1158.39,E2 1158.39} C_VEL
LIN {X 0,Y 601.886,Z 549.53,A -85,B 0,C 180,E1 1162.775,E2 1162.775} C_VEL
LIN {X 0,Y 602.035,Z 549.53,A -85,B 0,C 180,E1 1167.118,E2 1167.118} C_VEL
LIN {X 0,Y 602.131,Z 549.53,A -85,B 0,C 180,E1 1171.441,E2 1171.441} C_VEL
LIN {X 0,Y 602.171,Z 549.53,A -85,B 0,C 180,E1 1175.773,E2 1175.773} C_VEL
LIN {X 0,Y 601.833,Z 549.53,A -85,B 0,C 180,E1 1181.611,E2 1181.611} C_VEL
LIN {X 0,Y 601.855,Z 549.53,A -85,B 0,C 180,E1 1186.065,E2 1186.065} C_VEL
LIN {X 0,Y 601.733,Z 549.53,A -85,B 0,C 180,E1 1191.407,E2 1191.407} C_VEL
LIN {X 0,Y 601.985,Z 549.53,A -85,B 0,C 180,E1 1195.314,E2 1195.314} C_VEL
LIN {X 0,Y 601.72,Z 549.53,A -85,B 0,C 180,E1 1201.18,E2 1201.18} C_VEL
LIN {X 0,Y 601.763,Z 549.53,A -85,B 0,C 180,E1 1207.147,E2 1207.147} C_VEL
LIN {X 0,Y 601.568,Z 549.53,A -85,B 0,C 180,E1 1212.81,E2 1212.81} C_VEL
LIN {X 0,Y 601.963,Z 549.53,A -85,B 0,C 180,E1 1216.313,E2 1216.313} C_VEL
LIN {X 0,Y 603.546,Z 560.325,A -85,B 0,C 180,E1 1216.707,E2 1216.707} C_VEL
LIN {X 0,Y 603.404,Z 600.168,A -85,B 0,C 180,E1 1218.221,E2 1218.221} C_VEL
LIN {X 0,Y 603.119,Z 636.612,A -85,B 0,C 180,E1 1220.225,E2 1220.225} C_VEL
LIN {X 0,Y 602.828,Z 670.376,A -85,B 0,C 180,E1 1222.725,E2 1222.725} C_VEL
LIN {X 0,Y 602.539,Z 699.948,A -85,B 0,C 180,E1 1225.583,E2 1225.583} C_VEL
LIN {X 0,Y 602.376,Z 726.911,A -85,B 0,C 180,E1 1228.993,E2 1228.993} C_VEL
LIN {X 0,Y 602.272,Z 746.88,A -85,B 0,C 180,E1 1232.371,E2 1232.371} C_VEL
LIN {X 0,Y 602.228,Z 763.208,A -85,B 0,C 180,E1 1236.278,E2 1236.278} C_VEL
LIN {X 0,Y 602.132,Z 771.618,A -85,B 0,C 180,E1 1239.386,E2 1239.386} C_VEL
LIN {X 0,Y 602.077,Z 776.629,A -85,B 0,C 180,E1 1242.864,E2 1242.864} C_VEL
LIN {X 0,Y 602.224,Z 777.397,A -85,B 0,C 180,E1 1245.436,E2 1245.436} C_VEL
LIN {X 0,Y 602.206,Z 774.902,A -85,B 0,C 180,E1 1248.681,E2 1248.681} C_VEL
LIN {X 0,Y 602.22,Z 766.992,A -85,B 0,C 180,E1 1252.412,E2 1252.412} C_VEL
LIN {X 0,Y 602.254,Z 753.943,A -85,B 0,C 180,E1 1256.033,E2 1256.033} C_VEL
LIN {X 0,Y 602.139,Z 747.912,A -85,B 0,C 180,E1 1257.33,E2 1257.33} C_VEL
LIN {X 0,Y 598.331,Z 740.69,A -85,B 0,C 180,E1 1258.813,E2 1258.813} C_VEL
LIN {X 0,Y 594.47,Z 732.492,A -85,B 0,C 180,E1 1260.266,E2 1260.266} C_VEL
LIN {X 0,Y 594.725,Z 708.063,A -85,B 0,C 180,E1 1263.646,E2 1263.646} C_VEL
LIN {X 0,Y 595.161,Z 679.783,A -85,B 0,C 180,E1 1266.641,E2 1266.641} C_VEL
LIN {X 0,Y 595.666,Z 646.795,A -85,B 0,C 180,E1 1269.322,E2 1269.322} C_VEL
LIN {X 0,Y 596.222,Z 610.644,A -85,B 0,C 180,E1 1271.518,E2 1271.518} C_VEL
LIN {X 0,Y 596.655,Z 572.739,A -85,B 0,C 180,E1 1273.152,E2 1273.152} C_VEL
LIN {X 0,Y 596.049,Z 555.571,A -85,B 0,C 180,E1 1273.734,E2 1273.734} C_VEL
LIN {X 0,Y 594.25,Z 549.53,A -85,B 0,C 180,E1 1274.018,E2 1274.018} C_VEL
LIN {X 0,Y 593.938,Z 549.53,A -85,B 0,C 180,E1 1280.905,E2 1280.905} C_VEL
LIN {X 0,Y 593.933,Z 549.53,A -85,B 0,C 180,E1 1285.677,E2 1285.677} C_VEL
LIN {X 0,Y 593.842,Z 549.53,A -85,B 0,C 180,E1 1290.654,E2 1290.654} C_VEL
LIN {X 0,Y 593.802,Z 549.53,A -85,B 0,C 180,E1 1295.901,E2 1295.901} C_VEL
LIN {X 0,Y 593.786,Z 549.53,A -85,B 0,C 180,E1 1301.521,E2 1301.521} C_VEL
LIN {X 0,Y 593.675,Z 549.53,A -85,B 0,C 180,E1 1306.481,E2 1306.481} C_VEL
LIN {X 0,Y 593.697,Z 549.53,A -85,B 0,C 180,E1 1312.261,E2 1312.261} C_VEL
LIN {X 0,Y 593.974,Z 549.53,A -85,B 0,C 180,E1 1317.635,E2 1317.635} C_VEL
LIN {X 0,Y 594.105,Z 549.989,A -85,B 0,C 180,E1 1319.662,E2 1319.662} C_VEL
LIN {X 0,Y 596.604,Z 557.15,A -85,B 0,C 180,E1 1319.9,E2 1319.9} C_VEL
LIN {X 0,Y 596.832,Z 623.983,A -85,B 0,C 180,E1 1320.958,E2 1320.958} C_VEL
LIN {X 0,Y 596.55,Z 663.507,A -85,B 0,C 180,E1 1322.202,E2 1322.202} C_VEL
LIN {X 0,Y 596.026,Z 701.301,A -85,B 0,C 180,E1 1324.01,E2 1324.01} C_VEL
LIN {X 0,Y 595.499,Z 737.287,A -85,B 0,C 180,E1 1326.407,E2 1326.407} C_VEL
LIN {X 0,Y 595.027,Z 768.228,A -85,B 0,C 180,E1 1329.13,E2 1329.13} C_VEL
LIN {X 0,Y 594.671,Z 795.225,A -85,B 0,C 180,E1 1332.209,E2 1332.209} C_VEL
LIN {X 0,Y 594.462,Z 816.845,A -85,B 0,C 180,E1 1335.412,E2 1335.412} C_VEL
LIN {X 0,Y 594.292,Z 834.669,A -85,B 0,C 180,E1 1338.947,E2 1338.947} C_VEL
LIN {X 0,Y 594.233,Z 847.612,A -85,B 0,C 180,E1 1342.68,E2 1342.68} C_VEL
LIN {X 0,Y 594.134,Z 853.931,A -85,B 0,C 180,E1 1345.615,E2 1345.615} C_VEL
LIN {X 0,Y 594.163,Z 857.082,A -85,B 0,C 180,E1 1348.539,E2 1348.539} C_VEL
LIN {X 0,Y 594.298,Z 857.083,A -85,B 0,C 180,E1 1351.459,E2 1351.459} C_VEL
LIN {X 0,Y 594.393,Z 852.727,A -85,B 0,C 180,E1 1355.114,E2 1355.114} C_VEL
LIN {X 0,Y 594.304,Z 841.963,A -85,B 0,C 180,E1 1359.161,E2 1359.161} C_VEL
LIN {X 0,Y 594.4,Z 826.225,A -85,B 0,C 180,E1 1362.878,E2 1362.878} C_VEL
LIN {X 0,Y 594.569,Z 806.291,A -85,B 0,C 180,E1 1366.266,E2 1366.266} C_VEL
LIN {X 0,Y 594.902,Z 779.51,A -85,B 0,C 180,E1 1369.679,E2 1369.679} C_VEL
LIN {X 0,Y 595.291,Z 749.591,A -85,B 0,C 180,E1 1372.594,E2 1372.594} C_VEL
LIN {X 0,Y 595.785,Z 716.878,A -85,B 0,C 180,E1 1375.038,E2 1375.038} C_VEL
LIN {X 0,Y 596.301,Z 681.472,A -85,B 0,C 180,E1 1377.015,E2 1377.015} C_VEL
LIN {X 0,Y 596.714,Z 644.654,A -85,B 0,C 180,E1 1378.463,E2 1378.463} C_VEL
LIN {X 0,Y 596.906,Z 606.609,A -85,B 0,C 180,E1 1379.388,E2 1379.388} C_VEL
LIN {X 0,Y 595.998,Z 555.339,A -85,B 0,C 180,E1 1380.158,E2 1380.158} C_VEL
LIN {X 0,Y 593.949,Z 549.53,A -85,B 0,C 180,E1 1380.402,E2 1380.402} C_VEL
LIN {X 0,Y 593.829,Z 549.53,A -85,B 0,C 180,E1 1385.903,E2 1385.903} C_VEL
LIN {X 0,Y 593.795,Z 549.53,A -85,B 0,C 180,E1 1391.524,E2 1391.524} C_VEL
LIN {X 0,Y 593.67,Z 549.53,A -85,B 0,C 180,E1 1396.487,E2 1396.487} C_VEL
LIN {X 0,Y 593.674,Z 549.53,A -85,B 0,C 180,E1 1402.265,E2 1402.265} C_VEL
LIN {X 0,Y 593.863,Z 549.53,A -85,B 0,C 180,E1 1407.634,E2 1407.634} C_VEL
LIN {X 0,Y 593.746,Z 549.53,A -85,B 0,C 180,E1 1413.189,E2 1413.189} C_VEL
LIN {X 0,Y 593.754,Z 549.53,A -85,B 0,C 180,E1 1417.515,E2 1417.515} C_VEL
LIN {X 0,Y 594.006,Z 549.53,A -85,B 0,C 180,E1 1422.193,E2 1422.193} C_VEL
LIN {X 0,Y 593.919,Z 549.53,A -85,B 0,C 180,E1 1428.236,E2 1428.236} C_VEL
LIN {X 0,Y 593.979,Z 549.53,A -85,B 0,C 180,E1 1432.681,E2 1432.681} C_VEL
LIN {X 0,Y 594.061,Z 549.53,A -85,B 0,C 180,E1 1437.081,E2 1437.081} C_VEL
LIN {X 0,Y 594.199,Z 549.53,A -85,B 0,C 180,E1 1441.463,E2 1441.463} C_VEL
LIN {X 0,Y 594.072,Z 549.53,A -85,B 0,C 180,E1 1446.305,E2 1446.305} C_VEL
LIN {X 0,Y 593.858,Z 549.53,A -85,B 0,C 180,E1 1451.772,E2 1451.772} C_VEL
LIN {X 0,Y 593.89,Z 549.53,A -85,B 0,C 180,E1 1456.289,E2 1456.289} C_VEL
LIN {X 0,Y 593.929,Z 549.53,A -85,B 0,C 180,E1 1460.912,E2 1460.912} C_VEL
LIN {X 0,Y 593.929,Z 549.53,A -85,B 0,C 180,E1 1465.684,E2 1465.684} C_VEL
LIN {X 0,Y 593.772,Z 549.53,A -85,B 0,C 180,E1 1470.665,E2 1470.665} C_VEL
LIN {X 0,Y 593.812,Z 549.53,A -85,B 0,C 180,E1 1475.907,E2 1475.907} C_VEL
LIN {X 0,Y 593.757,Z 549.53,A -85,B 0,C 180,E1 1481.531,E2 1481.531} C_VEL
LIN {X 0,Y 593.665,Z 549.53,A -85,B 0,C 180,E1 1486.481,E2 1486.481} C_VEL
LIN {X 0,Y 593.666,Z 549.53,A -85,B 0,C 180,E1 1492.26,E2 1492.26} C_VEL
LIN {X 0,Y 593.858,Z 549.53,A -85,B 0,C 180,E1 1497.629,E2 1497.629} C_VEL
LIN {X 0,Y 593.737,Z 549.53,A -85,B 0,C 180,E1 1503.196,E2 1503.196} C_VEL
LIN {X 0,Y 593.766,Z 549.53,A -85,B 0,C 180,E1 1507.513,E2 1507.513} C_VEL
LIN {X 0,Y 594.047,Z 549.53,A -85,B 0,C 180,E1 1512.192,E2 1512.192} C_VEL
LIN {X 0,Y 593.933,Z 549.53,A -85,B 0,C 180,E1 1518.233,E2 1518.233} C_VEL
LIN {X 0,Y 593.996,Z 549.53,A -85,B 0,C 180,E1 1522.679,E2 1522.679} C_VEL
LIN {X 0,Y 594.128,Z 549.53,A -85,B 0,C 180,E1 1527.079,E2 1527.079} C_VEL
LIN {X 0,Y 594.221,Z 549.53,A -85,B 0,C 180,E1 1531.461,E2 1531.461} C_VEL
LIN {X 0,Y 594.084,Z 549.53,A -85,B 0,C 180,E1 1536.296,E2 1536.296} C_VEL
LIN {X 0,Y 593.896,Z 549.53,A -85,B 0,C 180,E1 1541.769,E2 1541.769} C_VEL
LIN {X 0,Y 593.908,Z 549.53,A -85,B 0,C 180,E1 1546.286,E2 1546.286} C_VEL
LIN {X 0,Y 593.945,Z 549.53,A -85,B 0,C 180,E1 1550.91,E2 1550.91} C_VEL
LIN {X 0,Y 593.968,Z 549.53,A -85,B 0,C 180,E1 1555.681,E2 1555.681} C_VEL
LIN {X 0,Y 593.842,Z 549.53,A -85,B 0,C 180,E1 1560.659,E2 1560.659} C_VEL
LIN {X 0,Y 593.829,Z 549.53,A -85,B 0,C 180,E1 1565.904,E2 1565.904} C_VEL
LIN {X 0,Y 593.679,Z 549.53,A -85,B 0,C 180,E1 1571.536,E2 1571.536} C_VEL
LIN {X 0,Y 593.938,Z 549.53,A -85,B 0,C 180,E1 1575.893,E2 1575.893} C_VEL
LIN {X 0,Y 596.531,Z 560.057,A -85,B 0,C 180,E1 1576.336,E2 1576.336} C_VEL
LIN {X 0,Y 596.251,Z 599.995,A -85,B 0,C 180,E1 1577.866,E2 1577.866} C_VEL
LIN {X 0,Y 595.779,Z 636.415,A -85,B 0,C 180,E1 1579.886,E2 1579.886} C_VEL
LIN {X 0,Y 595.33,Z 669.813,A -85,B 0,C 180,E1 1582.381,E2 1582.381} C_VEL
LIN {X 0,Y 594.892,Z 699.521,A -85,B 0,C 180,E1 1585.276,E2 1585.276} C_VEL
LIN {X 0,Y 594.579,Z 725.693,A -85,B 0,C 180,E1 1588.603,E2 1588.603} C_VEL
LIN {X 0,Y 594.412,Z 747.65,A -85,B 0,C 180,E1 1592.358,E2 1592.358} C_VEL
LIN {X 0,Y 594.326,Z 762.5,A -85,B 0,C 180,E1 1595.943,E2 1595.943} C_VEL
LIN {X 0,Y 594.229,Z 772.752,A -85,B 0,C 180,E1 1599.854,E2 1599.854} C_VEL
LIN {X 0,Y 594.261,Z 777.222,A -85,B 0,C 180,E1 1603.722,E2 1603.722} C_VEL
LIN {X 0,Y 594.253,Z 776.862,A -85,B 0,C 180,E1 1606.741,E2 1606.741} C_VEL
LIN {X 0,Y 594.168,Z 771.908,A -85,B 0,C 180,E1 1610.463,E2 1610.463} C_VEL
LIN {X 0,Y 594.227,Z 761.861,A -85,B 0,C 180,E1 1614.147,E2 1614.147} C_VEL
LIN {X 0,Y 594.32,Z 746.373,A -85,B 0,C 180,E1 1617.807,E2 1617.807} C_VEL
LIN {X 0,Y 594.47,Z 732.492,A -85,B 0,C 180,E1 1620.266,E2 1620.266} C_VEL
LIN {X 0,Y 590.655,Z 723.799,A -85,B 0,C 180,E1 1621.691,E2 1621.691} C_VEL
LIN {X 0,Y 586.952,Z 714.435,A -85,B 0,C 180,E1 1623.093,E2 1623.093} C_VEL
LIN {X 0,Y 587.533,Z 685.578,A -85,B 0,C 180,E1 1626.378,E2 1626.378} C_VEL
LIN {X 0,Y 588.159,Z 652.213,A -85,B 0,C 180,E1 1629.255,E2 1629.255} C_VEL
LIN {X 0,Y 588.903,Z 617.681,A -85,B 0,C 180,E1 1631.49,E2 1631.49} C_VEL
LIN {X 0,Y 589.512,Z 580.62,A -85,B 0,C 180,E1 1633.228,E2 1633.228} C_VEL
LIN {X 0,Y 589.002,Z 557.656,A -85,B 0,C 180,E1 1634.051,E2 1634.051} C_VEL
LIN {X 0,Y 586.323,Z 549.53,A -85,B 0,C 180,E1 1634.428,E2 1634.428} C_VEL
LIN {X 0,Y 585.958,Z 549.53,A -85,B 0,C 180,E1 1641.204,E2 1641.204} C_VEL
LIN {X 0,Y 585.971,Z 549.53,A -85,B 0,C 180,E1 1646.052,E2 1646.052} C_VEL
LIN {X 0,Y 585.789,Z 549.53,A -85,B 0,C 180,E1 1651.466,E2 1651.466} C_VEL
LIN {X 0,Y 585.844,Z 549.53,A -85,B 0,C 180,E1 1656.757,E2 1656.757} C_VEL
LIN {X 0,Y 585.9,Z 549.53,A -85,B 0,C 180,E1 1662.207,E2 1662.207} C_VEL
LIN {X 0,Y 585.703,Z 549.53,A -85,B 0,C 180,E1 1667.769,E2 1667.769} C_VEL
LIN {X 0,Y 585.708,Z 549.53,A -85,B 0,C 180,E1 1673.252,E2 1673.252} C_VEL
LIN {X 0,Y 586.061,Z 549.53,A -85,B 0,C 180,E1 1678.481,E2 1678.481} C_VEL
LIN {X 0,Y 586.2,Z 550.367,A -85,B 0,C 180,E1 1679.214,E2 1679.214} C_VEL
LIN {X 0,Y 589.73,Z 558.61,A -85,B 0,C 180,E1 1679.533,E2 1679.533} C_VEL
LIN {X 0,Y 589.931,Z 623.529,A -85,B 0,C 180,E1 1680.574,E2 1680.574} C_VEL
LIN {X 0,Y 589.488,Z 663.485,A -85,B 0,C 180,E1 1681.838,E2 1681.838} C_VEL
LIN {X 0,Y 588.776,Z 701.791,A -85,B 0,C 180,E1 1683.696,E2 1683.696} C_VEL
LIN {X 0,Y 588.07,Z 737.289,A -85,B 0,C 180,E1 1686.09,E2 1686.09} C_VEL
LIN {X 0,Y 587.462,Z 768.228,A -85,B 0,C 180,E1 1688.849,E2 1688.849} C_VEL
LIN {X 0,Y 586.926,Z 795.227,A -85,B 0,C 180,E1 1691.967,E2 1691.967} C_VEL
LIN {X 0,Y 586.625,Z 817.624,A -85,B 0,C 180,E1 1695.348,E2 1695.348} C_VEL
LIN {X 0,Y 586.421,Z 834.776,A -85,B 0,C 180,E1 1698.823,E2 1698.823} C_VEL
LIN {X 0,Y 586.336,Z 847.612,A -85,B 0,C 180,E1 1702.581,E2 1702.581} C_VEL
LIN {X 0,Y 586.234,Z 853.931,A -85,B 0,C 180,E1 1705.556,E2 1705.556} C_VEL
LIN {X 0,Y 586.27,Z 857.082,A -85,B 0,C 180,E1 1708.52,E2 1708.52} C_VEL
LIN {X 0,Y 586.392,Z 857.083,A -85,B 0,C 180,E1 1711.479,E2 1711.479} C_VEL
LIN {X 0,Y 586.487,Z 852.727,A -85,B 0,C 180,E1 1715.183,E2 1715.183} C_VEL
LIN {X 0,Y 586.431,Z 841.963,A -85,B 0,C 180,E1 1719.285,E2 1719.285} C_VEL
LIN {X 0,Y 586.555,Z 826.225,A -85,B 0,C 180,E1 1723.053,E2 1723.053} C_VEL
LIN {X 0,Y 586.777,Z 804.808,A -85,B 0,C 180,E1 1726.703,E2 1726.703} C_VEL
LIN {X 0,Y 587.201,Z 779.51,A -85,B 0,C 180,E1 1729.948,E2 1729.948} C_VEL
LIN {X 0,Y 587.79,Z 749.847,A -85,B 0,C 180,E1 1732.876,E2 1732.876} C_VEL
LIN {X 0,Y 588.466,Z 716.375,A -85,B 0,C 180,E1 1735.405,E2 1735.405} C_VEL
LIN {X 0,Y 589.153,Z 681.883,A -85,B 0,C 180,E1 1737.35,E2 1737.35} C_VEL
LIN {X 0,Y 589.727,Z 645.089,A -85,B 0,C 180,E1 1738.817,E2 1738.817} C_VEL
LIN {X 0,Y 590.014,Z 607.486,A -85,B 0,C 180,E1 1739.751,E2 1739.751} C_VEL
LIN {X 0,Y 589.178,Z 557.954,A -85,B 0,C 180,E1 1740.508,E2 1740.508} C_VEL
LIN {X 0,Y 585.945,Z 549.53,A -85,B 0,C 180,E1 1740.9,E2 1740.9} C_VEL
LIN {X 0,Y 585.849,Z 549.53,A -85,B 0,C 180,E1 1746.766,E2 1746.766} C_VEL
LIN {X 0,Y 585.903,Z 549.53,A -85,B 0,C 180,E1 1752.212,E2 1752.212} C_VEL
LIN {X 0,Y 585.701,Z 549.53,A -85,B 0,C 180,E1 1757.775,E2 1757.775} C_VEL
LIN {X 0,Y 585.691,Z 549.53,A -85,B 0,C 180,E1 1763.261,E2 1763.261} C_VEL
LIN {X 0,Y 585.901,Z 549.53,A -85,B 0,C 180,E1 1768.513,E2 1768.513} C_VEL
LIN {X 0,Y 585.81,Z 549.53,A -85,B 0,C 180,E1 1773.94,E2 1773.94} C_VEL
LIN {X 0,Y 585.772,Z 549.53,A -85,B 0,C 180,E1 1778.789,E2 1778.789} C_VEL
LIN {X 0,Y 585.931,Z 549.53,A -85,B 0,C 180,E1 1783.49,E2 1783.49} C_VEL
LIN {X 0,Y 586.039,Z 549.53,A -85,B 0,C 180,E1 1788.075,E2 1788.075} C_VEL
LIN {X 0,Y 586.073,Z 549.53,A -85,B 0,C 180,E1 1792.582,E2 1792.582} C_VEL
LIN {X 0,Y 586.169,Z 549.53,A -85,B 0,C 180,E1 1797.042,E2 1797.042} C_VEL
LIN {X 0,Y 586.298,Z 549.53,A -85,B 0,C 180,E1 1801.483,E2 1801.483} C_VEL
LIN {X 0,Y 586.305,Z 549.53,A -85,B 0,C 180,E1 1805.932,E2 1805.932} C_VEL
LIN {X 0,Y 585.927,Z 549.53,A -85,B 0,C 180,E1 1811.933,E2 1811.933} C_VEL
LIN {X 0,Y 585.86,Z 549.53,A -85,B 0,C 180,E1 1817.021,E2 1817.021} C_VEL
LIN {X 0,Y 585.913,Z 549.53,A -85,B 0,C 180,E1 1821.523,E2 1821.523} C_VEL
LIN {X 0,Y 585.968,Z 549.53,A -85,B 0,C 180,E1 1826.059,E2 1826.059} C_VEL
LIN {X 0,Y 585.748,Z 549.53,A -85,B 0,C 180,E1 1831.462,E2 1831.462} C_VEL
LIN {X 0,Y 585.85,Z 549.53,A -85,B 0,C 180,E1 1836.76,E2 1836.76} C_VEL
LIN {X 0,Y 585.874,Z 549.53,A -85,B 0,C 180,E1 1842.218,E2 1842.218} C_VEL
LIN {X 0,Y 585.696,Z 549.53,A -85,B 0,C 180,E1 1847.77,E2 1847.77} C_VEL
LIN {X 0,Y 585.686,Z 549.53,A -85,B 0,C 180,E1 1853.266,E2 1853.266} C_VEL
LIN {X 0,Y 585.877,Z 549.53,A -85,B 0,C 180,E1 1858.522,E2 1858.522} C_VEL
LIN {X 0,Y 585.799,Z 549.53,A -85,B 0,C 180,E1 1863.936,E2 1863.936} C_VEL
LIN {X 0,Y 585.79,Z 549.53,A -85,B 0,C 180,E1 1868.787,E2 1868.787} C_VEL
LIN {X 0,Y 585.971,Z 549.53,A -85,B 0,C 180,E1 1873.488,E2 1873.488} C_VEL
LIN {X 0,Y 586.055,Z 549.53,A -85,B 0,C 180,E1 1878.073,E2 1878.073} C_VEL
LIN {X 0,Y 586.089,Z 549.53,A -85,B 0,C 180,E1 1882.579,E2 1882.579} C_VEL
LIN {X 0,Y 586.234,Z 549.53,A -85,B 0,C 180,E1 1887.04,E2 1887.04} C_VEL
LIN {X 0,Y 586.319,Z 549.53,A -85,B 0,C 180,E1 1891.48,E2 1891.48} C_VEL
LIN {X 0,Y 586.308,Z 549.53,A -85,B 0,C 180,E1 1895.93,E2 1895.93} C_VEL
LIN {X 0,Y 585.994,Z 549.53,A -85,B 0,C 180,E1 1901.93,E2 1901.93} C_VEL
LIN {X 0,Y 585.9,Z 549.53,A -85,B 0,C 180,E1 1907.026,E2 1907.026} C_VEL
LIN {X 0,Y 585.934,Z 549.53,A -85,B 0,C 180,E1 1911.522,E2 1911.522} C_VEL
LIN {X 0,Y 586.004,Z 549.53,A -85,B 0,C 180,E1 1916.056,E2 1916.056} C_VEL
LIN {X 0,Y 585.802,Z 549.53,A -85,B 0,C 180,E1 1921.466,E2 1921.466} C_VEL
LIN {X 0,Y 585.876,Z 549.53,A -85,B 0,C 180,E1 1926.759,E2 1926.759} C_VEL
LIN {X 0,Y 585.747,Z 549.53,A -85,B 0,C 180,E1 1932.227,E2 1932.227} C_VEL
LIN {X 0,Y 585.905,Z 549.776,A -85,B 0,C 180,E1 1935.472,E2 1935.472} C_VEL
LIN {X 0,Y 589.556,Z 562.353,A -85,B 0,C 180,E1 1936.039,E2 1936.039} C_VEL
LIN {X 0,Y 589.103,Z 601.342,A -85,B 0,C 180,E1 1937.575,E2 1937.575} C_VEL
LIN {X 0,Y 588.445,Z 636.928,A -85,B 0,C 180,E1 1939.585,E2 1939.585} C_VEL
LIN {X 0,Y 587.818,Z 670.652,A -85,B 0,C 180,E1 1942.149,E2 1942.149} C_VEL
LIN {X 0,Y 587.227,Z 700.388,A -85,B 0,C 180,E1 1945.105,E2 1945.105} C_VEL
LIN {X 0,Y 586.783,Z 725.673,A -85,B 0,C 180,E1 1948.376,E2 1948.376} C_VEL
LIN {X 0,Y 586.522,Z 747.107,A -85,B 0,C 180,E1 1952.074,E2 1952.074} C_VEL
LIN {X 0,Y 586.429,Z 761.716,A -85,B 0,C 180,E1 1955.598,E2 1955.598} C_VEL
LIN {X 0,Y 586.318,Z 772.375,A -85,B 0,C 180,E1 1959.595,E2 1959.595} C_VEL
LIN {X 0,Y 586.32,Z 777.104,A -85,B 0,C 180,E1 1963.495,E2 1963.495} C_VEL
LIN {X 0,Y 586.356,Z 777.005,A -85,B 0,C 180,E1 1966.559,E2 1966.559} C_VEL
LIN {X 0,Y 586.27,Z 772.338,A -85,B 0,C 180,E1 1970.333,E2 1970.333} C_VEL
LIN {X 0,Y 586.35,Z 762.575,A -85,B 0,C 180,E1 1974.069,E2 1974.069} C_VEL
LIN {X 0,Y 586.463,Z 747.397,A -85,B 0,C 180,E1 1977.778,E2 1977.778} C_VEL
LIN {X 0,Y 586.737,Z 726.086,A -85,B 0,C 180,E1 1981.476,E2 1981.476} C_VEL
LIN {X 0,Y 586.952,Z 714.435,A -85,B 0,C 180,E1 1983.093,E2 1983.093} C_VEL
LIN {X 0,Y 583.269,Z 704.517,A -85,B 0,C 180,E1 1984.463,E2 1984.463} C_VEL
LIN {X 0,Y 579.738,Z 693.962,A -85,B 0,C 180,E1 1985.799,E2 1985.799} C_VEL
LIN {X 0,Y 580.538,Z 662.01,A -85,B 0,C 180,E1 1988.81,E2 1988.81} C_VEL
LIN {X 0,Y 581.395,Z 627.651,A -85,B 0,C 180,E1 1991.26,E2 1991.26} C_VEL
LIN {X 0,Y 582.17,Z 590.857,A -85,B 0,C 180,E1 1993.182,E2 1993.182} C_VEL
LIN {X 0,Y 582.118,Z 560.602,A -85,B 0,C 180,E1 1994.334,E2 1994.334} C_VEL
LIN {X 0,Y 578.3,Z 549.53,A -85,B 0,C 180,E1 1994.965,E2 1994.965} C_VEL
LIN {X 0,Y 578.029,Z 549.53,A -85,B 0,C 180,E1 2001.509,E2 2001.509} C_VEL
LIN {X 0,Y 577.913,Z 549.53,A -85,B 0,C 180,E1 2007.03,E2 2007.03} C_VEL
LIN {X 0,Y 577.88,Z 549.53,A -85,B 0,C 180,E1 2011.597,E2 2011.597} C_VEL
LIN {X 0,Y 577.93,Z 549.53,A -85,B 0,C 180,E1 2017.048,E2 2017.048} C_VEL
LIN {X 0,Y 577.959,Z 549.53,A -85,B 0,C 180,E1 2022.925,E2 2022.925} C_VEL
LIN {X 0,Y 577.811,Z 549.53,A -85,B 0,C 180,E1 2029.073,E2 2029.073} C_VEL
LIN {X 0,Y 577.882,Z 549.53,A -85,B 0,C 180,E1 2034.801,E2 2034.801} C_VEL
LIN {X 0,Y 578.23,Z 550.18,A -85,B 0,C 180,E1 2038.74,E2 2038.74} C_VEL
LIN {X 0,Y 582.886,Z 561.326,A -85,B 0,C 180,E1 2039.174,E2 2039.174} C_VEL
LIN {X 0,Y 583.014,Z 624.902,A -85,B 0,C 180,E1 2040.226,E2 2040.226} C_VEL
LIN {X 0,Y 582.458,Z 663.422,A -85,B 0,C 180,E1 2041.465,E2 2041.465} C_VEL
LIN {X 0,Y 581.54,Z 701.695,A -85,B 0,C 180,E1 2043.337,E2 2043.337} C_VEL
LIN {X 0,Y 580.683,Z 736.432,A -85,B 0,C 180,E1 2045.697,E2 2045.697} C_VEL
LIN {X 0,Y 579.842,Z 768.228,A -85,B 0,C 180,E1 2048.557,E2 2048.557} C_VEL
LIN {X 0,Y 579.211,Z 795.228,A -85,B 0,C 180,E1 2051.718,E2 2051.718} C_VEL
LIN {X 0,Y 578.816,Z 817.883,A -85,B 0,C 180,E1 2055.192,E2 2055.192} C_VEL
LIN {X 0,Y 578.527,Z 834.776,A -85,B 0,C 180,E1 2058.668,E2 2058.668} C_VEL
LIN {X 0,Y 578.443,Z 847.612,A -85,B 0,C 180,E1 2062.479,E2 2062.479} C_VEL
LIN {X 0,Y 578.336,Z 853.931,A -85,B 0,C 180,E1 2065.495,E2 2065.495} C_VEL
LIN {X 0,Y 578.368,Z 857.082,A -85,B 0,C 180,E1 2068.499,E2 2068.499} C_VEL
LIN {X 0,Y 578.487,Z 857.084,A -85,B 0,C 180,E1 2071.499,E2 2071.499} C_VEL
LIN {X 0,Y 578.588,Z 852.753,A -85,B 0,C 180,E1 2075.24,E2 2075.24} C_VEL
LIN {X 0,Y 578.536,Z 843.212,A -85,B 0,C 180,E1 2079.034,E2 2079.034} C_VEL
LIN {X 0,Y 578.708,Z 828.083,A -85,B 0,C 180,E1 2082.848,E2 2082.848} C_VEL
LIN {X 0,Y 578.985,Z 806.288,A -85,B 0,C 180,E1 2086.717,E2 2086.717} C_VEL
LIN {X 0,Y 579.551,Z 779.921,A -85,B 0,C 180,E1 2090.176,E2 2090.176} C_VEL
LIN {X 0,Y 580.322,Z 749.996,A -85,B 0,C 180,E1 2093.175,E2 2093.175} C_VEL
LIN {X 0,Y 581.143,Z 716.945,A -85,B 0,C 180,E1 2095.71,E2 2095.71} C_VEL
LIN {X 0,Y 582.044,Z 680.915,A -85,B 0,C 180,E1 2097.76,E2 2097.76} C_VEL
LIN {X 0,Y 582.769,Z 644.546,A -85,B 0,C 180,E1 2099.212,E2 2099.212} C_VEL
LIN {X 0,Y 583.173,Z 607.206,A -85,B 0,C 180,E1 2100.141,E2 2100.141} C_VEL
LIN {X 0,Y 582.514,Z 560.778,A -85,B 0,C 180,E1 2100.855,E2 2100.855} C_VEL
LIN {X 0,Y 577.961,Z 549.53,A -85,B 0,C 180,E1 2101.299,E2 2101.299} C_VEL
LIN {X 0,Y 577.93,Z 549.53,A -85,B 0,C 180,E1 2107.052,E2 2107.052} C_VEL
LIN {X 0,Y 577.976,Z 549.53,A -85,B 0,C 180,E1 2112.928,E2 2112.928} C_VEL
LIN {X 0,Y 577.805,Z 549.53,A -85,B 0,C 180,E1 2119.079,E2 2119.079} C_VEL
LIN {X 0,Y 577.837,Z 549.53,A -85,B 0,C 180,E1 2124.804,E2 2124.804} C_VEL
LIN {X 0,Y 577.958,Z 549.53,A -85,B 0,C 180,E1 2130.154,E2 2130.154} C_VEL
LIN {X 0,Y 577.922,Z 549.53,A -85,B 0,C 180,E1 2135.222,E2 2135.222} C_VEL
LIN {X 0,Y 577.981,Z 549.53,A -85,B 0,C 180,E1 2140.568,E2 2140.568} C_VEL
LIN {X 0,Y 578.181,Z 549.53,A -85,B 0,C 180,E1 2146.372,E2 2146.372} C_VEL
LIN {X 0,Y 578.173,Z 549.53,A -85,B 0,C 180,E1 2152.48,E2 2152.48} C_VEL
LIN {X 0,Y 578.26,Z 549.53,A -85,B 0,C 180,E1 2157.001,E2 2157.001} C_VEL
LIN {X 0,Y 578.388,Z 549.53,A -85,B 0,C 180,E1 2161.503,E2 2161.503} C_VEL
LIN {X 0,Y 578.37,Z 549.53,A -85,B 0,C 180,E1 2166.014,E2 2166.014} C_VEL
LIN {X 0,Y 578.004,Z 549.53,A -85,B 0,C 180,E1 2172.099,E2 2172.099} C_VEL
LIN {X 0,Y 578.016,Z 549.53,A -85,B 0,C 180,E1 2176.749,E2 2176.749} C_VEL
LIN {X 0,Y 578.024,Z 549.53,A -85,B 0,C 180,E1 2181.516,E2 2181.516} C_VEL
LIN {X 0,Y 577.906,Z 549.53,A -85,B 0,C 180,E1 2187.031,E2 2187.031} C_VEL
LIN {X 0,Y 577.814,Z 549.53,A -85,B 0,C 180,E1 2193.018,E2 2193.018} C_VEL
LIN {X 0,Y 577.9,Z 549.53,A -85,B 0,C 180,E1 2198.189,E2 2198.189} C_VEL
LIN {X 0,Y 577.946,Z 549.53,A -85,B 0,C 180,E1 2202.935,E2 2202.935} C_VEL
LIN {X 0,Y 577.799,Z 549.53,A -85,B 0,C 180,E1 2209.074,E2 2209.074} C_VEL
LIN {X 0,Y 577.838,Z 549.53,A -85,B 0,C 180,E1 2214.8,E2 2214.8} C_VEL
LIN {X 0,Y 577.93,Z 549.53,A -85,B 0,C 180,E1 2220.149,E2 2220.149} C_VEL
LIN {X 0,Y 577.921,Z 549.53,A -85,B 0,C 180,E1 2225.218,E2 2225.218} C_VEL
LIN {X 0,Y 578.011,Z 549.53,A -85,B 0,C 180,E1 2230.566,E2 2230.566} C_VEL
LIN {X 0,Y 578.202,Z 549.53,A -85,B 0,C 180,E1 2236.369,E2 2236.369} C_VEL
LIN {X 0,Y 578.19,Z 549.53,A -85,B 0,C 180,E1 2242.477,E2 2242.477} C_VEL
LIN {X 0,Y 578.326,Z 549.53,A -85,B 0,C 180,E1 2246.999,E2 2246.999} C_VEL
LIN {X 0,Y 578.409,Z 549.53,A -85,B 0,C 180,E1 2251.501,E2 2251.501} C_VEL
LIN {X 0,Y 578.384,Z 549.53,A -85,B 0,C 180,E1 2256.011,E2 2256.011} C_VEL
LIN {X 0,Y 578.067,Z 549.53,A -85,B 0,C 180,E1 2262.096,E2 2262.096} C_VEL
LIN {X 0,Y 578.046,Z 549.53,A -85,B 0,C 180,E1 2266.746,E2 2266.746} C_VEL
LIN {X 0,Y 578.045,Z 549.53,A -85,B 0,C 180,E1 2271.513,E2 2271.513} C_VEL
LIN {X 0,Y 577.945,Z 549.53,A -85,B 0,C 180,E1 2277.033,E2 2277.033} C_VEL
LIN {X 0,Y 577.896,Z 549.53,A -85,B 0,C 180,E1 2281.601,E2 2281.601} C_VEL
LIN {X 0,Y 577.96,Z 549.53,A -85,B 0,C 180,E1 2287.052,E2 2287.052} C_VEL
LIN {X 0,Y 577.779,Z 549.53,A -85,B 0,C 180,E1 2292.948,E2 2292.948} C_VEL
LIN {X 0,Y 577.886,Z 549.926,A -85,B 0,C 180,E1 2295.025,E2 2295.025} C_VEL
LIN {X 0,Y 582.573,Z 564.429,A -85,B 0,C 180,E1 2295.726,E2 2295.726} C_VEL
LIN {X 0,Y 581.949,Z 603.063,A -85,B 0,C 180,E1 2297.295,E2 2297.295} C_VEL
LIN {X 0,Y 581.085,Z 639.697,A -85,B 0,C 180,E1 2299.429,E2 2299.429} C_VEL
LIN {X 0,Y 580.247,Z 673.657,A -85,B 0,C 180,E1 2302.101,E2 2302.101} C_VEL
LIN {X 0,Y 579.478,Z 703.448,A -85,B 0,C 180,E1 2305.184,E2 2305.184} C_VEL
LIN {X 0,Y 578.973,Z 728.768,A -85,B 0,C 180,E1 2308.625,E2 2308.625} C_VEL
LIN {X 0,Y 578.712,Z 749.439,A -85,B 0,C 180,E1 2312.402,E2 2312.402} C_VEL
LIN {X 0,Y 578.54,Z 762.956,A -85,B 0,C 180,E1 2315.836,E2 2315.836} C_VEL
LIN {X 0,Y 578.415,Z 771.926,A -85,B 0,C 180,E1 2319.303,E2 2319.303} C_VEL
LIN {X 0,Y 578.393,Z 776.963,A -85,B 0,C 180,E1 2323.262,E2 2323.262} C_VEL
LIN {X 0,Y 578.438,Z 777.147,A -85,B 0,C 180,E1 2326.372,E2 2326.372} C_VEL
LIN {X 0,Y 578.387,Z 772.742,A -85,B 0,C 180,E1 2330.2,E2 2330.2} C_VEL
LIN {X 0,Y 578.458,Z 763.007,A -85,B 0,C 180,E1 2334.059,E2 2334.059} C_VEL
LIN {X 0,Y 578.625,Z 748.357,A -85,B 0,C 180,E1 2337.747,E2 2337.747} C_VEL
LIN {X 0,Y 578.881,Z 728.64,A -85,B 0,C 180,E1 2341.308,E2 2341.308} C_VEL
LIN {X 0,Y 579.473,Z 702.256,A -85,B 0,C 180,E1 2344.868,E2 2344.868} C_VEL
LIN {X 0,Y 579.738,Z 693.962,A -85,B 0,C 180,E1 2345.799,E2 2345.799} C_VEL
LIN {X 0,Y 576.272,Z 682.882,A -85,B 0,C 180,E1 2347.103,E2 2347.103} C_VEL
LIN {X 0,Y 572.821,Z 671.103,A -85,B 0,C 180,E1 2348.353,E2 2348.353} C_VEL
LIN {X 0,Y 573.853,Z 638.232,A -85,B 0,C 180,E1 2350.928,E2 2350.928} C_VEL
LIN {X 0,Y 574.909,Z 602.216,A -85,B 0,C 180,E1 2353.026,E2 2353.026} C_VEL
LIN {X 0,Y 575.115,Z 562.996,A -85,B 0,C 180,E1 2354.649,E2 2354.649} C_VEL
LIN {X 0,Y 570.273,Z 549.53,A -85,B 0,C 180,E1 2355.393,E2 2355.393} C_VEL
LIN {X 0,Y 570.1,Z 549.53,A -85,B 0,C 180,E1 2361.823,E2 2361.823} C_VEL
LIN {X 0,Y 570.043,Z 549.53,A -85,B 0,C 180,E1 2366.837,E2 2366.837} C_VEL
LIN {X 0,Y 569.919,Z 549.53,A -85,B 0,C 180,E1 2372.09,E2 2372.09} C_VEL
LIN {X 0,Y 570.024,Z 549.53,A -85,B 0,C 180,E1 2377.65,E2 2377.65} C_VEL
LIN {X 0,Y 569.965,Z 549.53,A -85,B 0,C 180,E1 2383.677,E2 2383.677} C_VEL
LIN {X 0,Y 569.839,Z 549.53,A -85,B 0,C 180,E1 2388.374,E2 2388.374} C_VEL
LIN {X 0,Y 569.929,Z 549.53,A -85,B 0,C 180,E1 2394.235,E2 2394.235} C_VEL
LIN {X 0,Y 570.281,Z 550.15,A -85,B 0,C 180,E1 2398.254,E2 2398.254} C_VEL
LIN {X 0,Y 576.215,Z 563.951,A -85,B 0,C 180,E1 2398.815,E2 2398.815} C_VEL
LIN {X 0,Y 576.157,Z 624.337,A -85,B 0,C 180,E1 2399.82,E2 2399.82} C_VEL
LIN {X 0,Y 575.444,Z 663.473,A -85,B 0,C 180,E1 2401.087,E2 2401.087} C_VEL
LIN {X 0,Y 574.356,Z 701.222,A -85,B 0,C 180,E1 2402.947,E2 2402.947} C_VEL
LIN {X 0,Y 573.287,Z 736.425,A -85,B 0,C 180,E1 2405.363,E2 2405.363} C_VEL
LIN {X 0,Y 572.246,Z 768.227,A -85,B 0,C 180,E1 2408.258,E2 2408.258} C_VEL
LIN {X 0,Y 571.507,Z 795.229,A -85,B 0,C 180,E1 2411.463,E2 2411.463} C_VEL
LIN {X 0,Y 571.004,Z 817.883,A -85,B 0,C 180,E1 2414.984,E2 2414.984} C_VEL
LIN {X 0,Y 570.684,Z 835.832,A -85,B 0,C 180,E1 2418.775,E2 2418.775} C_VEL
LIN {X 0,Y 570.553,Z 847.612,A -85,B 0,C 180,E1 2422.375,E2 2422.375} C_VEL
LIN {X 0,Y 570.468,Z 853.931,A -85,B 0,C 180,E1 2425.432,E2 2425.432} C_VEL
LIN {X 0,Y 570.478,Z 857.083,A -85,B 0,C 180,E1 2428.479,E2 2428.479} C_VEL
LIN {X 0,Y 570.587,Z 857.084,A -85,B 0,C 180,E1 2431.52,E2 2431.52} C_VEL
LIN {X 0,Y 570.695,Z 852.941,A -85,B 0,C 180,E1 2435.195,E2 2435.195} C_VEL
LIN {X 0,Y 570.648,Z 843.212,A -85,B 0,C 180,E1 2439.159,E2 2439.159} C_VEL
LIN {X 0,Y 570.871,Z 828.084,A -85,B 0,C 180,E1 2443.028,E2 2443.028} C_VEL
LIN {X 0,Y 571.204,Z 807.569,A -85,B 0,C 180,E1 2446.753,E2 2446.753} C_VEL
LIN {X 0,Y 571.889,Z 781.007,A -85,B 0,C 180,E1 2450.333,E2 2450.333} C_VEL
LIN {X 0,Y 572.8,Z 751.538,A -85,B 0,C 180,E1 2453.358,E2 2453.358} C_VEL
LIN {X 0,Y 573.812,Z 718.533,A -85,B 0,C 180,E1 2455.953,E2 2455.953} C_VEL
LIN {X 0,Y 574.879,Z 684.108,A -85,B 0,C 180,E1 2457.976,E2 2457.976} C_VEL
LIN {X 0,Y 575.783,Z 647.227,A -85,B 0,C 180,E1 2459.513,E2 2459.513} C_VEL
LIN {X 0,Y 576.345,Z 608.067,A -85,B 0,C 180,E1 2460.521,E2 2460.521} C_VEL
LIN {X 0,Y 575.675,Z 562.955,A -85,B 0,C 180,E1 2461.232,E2 2461.232} C_VEL
LIN {X 0,Y 570,Z 549.53,A -85,B 0,C 180,E1 2461.797,E2 2461.797} C_VEL
LIN {X 0,Y 570.015,Z 549.53,A -85,B 0,C 180,E1 2467.655,E2 2467.655} C_VEL
LIN {X 0,Y 569.97,Z 549.53,A -85,B 0,C 180,E1 2473.682,E2 2473.682} C_VEL
LIN {X 0,Y 569.834,Z 549.53,A -85,B 0,C 180,E1 2478.38,E2 2478.38} C_VEL
LIN {X 0,Y 569.897,Z 549.53,A -85,B 0,C 180,E1 2484.239,E2 2484.239} C_VEL
LIN {X 0,Y 570.065,Z 549.53,A -85,B 0,C 180,E1 2489.698,E2 2489.698} C_VEL
LIN {X 0,Y 569.969,Z 549.53,A -85,B 0,C 180,E1 2494.852,E2 2494.852} C_VEL
LIN {X 0,Y 570.004,Z 549.53,A -85,B 0,C 180,E1 2499.803,E2 2499.803} C_VEL
LIN {X 0,Y 570.033,Z 549.53,A -85,B 0,C 180,E1 2504.601,E2 2504.601} C_VEL
LIN {X 0,Y 570.129,Z 549.53,A -85,B 0,C 180,E1 2509.29,E2 2509.29} C_VEL
LIN {X 0,Y 570.161,Z 549.53,A -85,B 0,C 180,E1 2513.906,E2 2513.906} C_VEL
LIN {X 0,Y 570.183,Z 549.53,A -85,B 0,C 180,E1 2518.482,E2 2518.482} C_VEL
LIN {X 0,Y 570.196,Z 549.53,A -85,B 0,C 180,E1 2523.047,E2 2523.047} C_VEL
LIN {X 0,Y 570.13,Z 549.53,A -85,B 0,C 180,E1 2527.633,E2 2527.633} C_VEL
LIN {X 0,Y 570.1,Z 549.53,A -85,B 0,C 180,E1 2532.27,E2 2532.27} C_VEL
LIN {X 0,Y 570.079,Z 549.53,A -85,B 0,C 180,E1 2537.039,E2 2537.039} C_VEL
LIN {X 0,Y 570.073,Z 549.53,A -85,B 0,C 180,E1 2541.831,E2 2541.831} C_VEL
LIN {X 0,Y 570.037,Z 549.53,A -85,B 0,C 180,E1 2546.845,E2 2546.845} C_VEL
LIN {X 0,Y 569.904,Z 549.53,A -85,B 0,C 180,E1 2552.099,E2 2552.099} C_VEL
LIN {X 0,Y 569.99,Z 549.53,A -85,B 0,C 180,E1 2557.661,E2 2557.661} C_VEL
LIN {X 0,Y 569.95,Z 549.53,A -85,B 0,C 180,E1 2563.687,E2 2563.687} C_VEL
LIN {X 0,Y 569.833,Z 549.53,A -85,B 0,C 180,E1 2568.375,E2 2568.375} C_VEL
LIN {X 0,Y 569.896,Z 549.53,A -85,B 0,C 180,E1 2574.234,E2 2574.234} C_VEL
LIN {X 0,Y 570.041,Z 549.53,A -85,B 0,C 180,E1 2579.693,E2 2579.693} C_VEL
LIN {X 0,Y 569.965,Z 549.53,A -85,B 0,C 180,E1 2584.848,E2 2584.848} C_VEL
LIN {X 0,Y 570.031,Z 549.53,A -85,B 0,C 180,E1 2589.801,E2 2589.801} C_VEL
LIN {X 0,Y 570.069,Z 549.53,A -85,B 0,C 180,E1 2594.598,E2 2594.598} C_VEL
LIN {X 0,Y 570.123,Z 549.53,A -85,B 0,C 180,E1 2599.306,E2 2599.306} C_VEL
LIN {X 0,Y 570.19,Z 549.53,A -85,B 0,C 180,E1 2603.904,E2 2603.904} C_VEL
LIN {X 0,Y 570.232,Z 549.53,A -85,B 0,C 180,E1 2608.479,E2 2608.479} C_VEL
LIN {X 0,Y 570.209,Z 549.53,A -85,B 0,C 180,E1 2613.045,E2 2613.045} C_VEL
LIN {X 0,Y 570.15,Z 549.53,A -85,B 0,C 180,E1 2617.631,E2 2617.631} C_VEL
LIN {X 0,Y 570.156,Z 549.53,A -85,B 0,C 180,E1 2622.266,E2 2622.266} C_VEL
LIN {X 0,Y 570.121,Z 549.53,A -85,B 0,C 180,E1 2627.044,E2 2627.044} C_VEL
LIN {X 0,Y 570.122,Z 549.53,A -85,B 0,C 180,E1 2631.827,E2 2631.827} C_VEL
LIN {X 0,Y 570.075,Z 549.53,A -85,B 0,C 180,E1 2636.841,E2 2636.841} C_VEL
LIN {X 0,Y 569.943,Z 549.53,A -85,B 0,C 180,E1 2642.094,E2 2642.094} C_VEL
LIN {X 0,Y 570.019,Z 549.53,A -85,B 0,C 180,E1 2647.657,E2 2647.657} C_VEL
LIN {X 0,Y 569.832,Z 549.53,A -85,B 0,C 180,E1 2653.697,E2 2653.697} C_VEL
LIN {X 0,Y 569.933,Z 550.012,A -85,B 0,C 180,E1 2654.565,E2 2654.565} C_VEL
LIN {X 0,Y 575.61,Z 566.348,A -85,B 0,C 180,E1 2655.401,E2 2655.401} C_VEL
LIN {X 0,Y 574.776,Z 606.164,A -85,B 0,C 180,E1 2657.076,E2 2657.076} C_VEL
LIN {X 0,Y 573.69,Z 643.49,A -85,B 0,C 180,E1 2659.342,E2 2659.342} C_VEL
LIN {X 0,Y 572.634,Z 677.771,A -85,B 0,C 180,E1 2662.172,E2 2662.172} C_VEL
LIN {X 0,Y 571.748,Z 706.359,A -85,B 0,C 180,E1 2665.269,E2 2665.269} C_VEL
LIN {X 0,Y 571.164,Z 730.119,A -85,B 0,C 180,E1 2668.615,E2 2668.615} C_VEL
LIN {X 0,Y 570.864,Z 750.305,A -85,B 0,C 180,E1 2672.418,E2 2672.418} C_VEL
LIN {X 0,Y 570.633,Z 763.848,A -85,B 0,C 180,E1 2676.005,E2 2676.005} C_VEL
LIN {X 0,Y 570.507,Z 773.045,A -85,B 0,C 180,E1 2679.815,E2 2679.815} C_VEL
LIN {X 0,Y 570.459,Z 776.822,A -85,B 0,C 180,E1 2683.022,E2 2683.022} C_VEL
LIN {X 0,Y 570.532,Z 777.245,A -85,B 0,C 180,E1 2686.179,E2 2686.179} C_VEL
LIN {X 0,Y 570.512,Z 773.093,A -85,B 0,C 180,E1 2690.064,E2 2690.064} C_VEL
LIN {X 0,Y 570.572,Z 763.853,A -85,B 0,C 180,E1 2693.904,E2 2693.904} C_VEL
LIN {X 0,Y 570.745,Z 751.017,A -85,B 0,C 180,E1 2697.336,E2 2697.336} C_VEL
LIN {X 0,Y 571.063,Z 732.277,A -85,B 0,C 180,E1 2700.946,E2 2700.946} C_VEL
LIN {X 0,Y 571.673,Z 708.599,A -85,B 0,C 180,E1 2704.364,E2 2704.364} C_VEL
LIN {X 0,Y 572.548,Z 679.277,A -85,B 0,C 180,E1 2707.595,E2 2707.595} C_VEL
LIN {X 0,Y 572.821,Z 671.103,A -85,B 0,C 180,E1 2708.353,E2 2708.353} C_VEL
LIN {X 0,Y 569.274,Z 663.459,A -85,B 0,C 180,E1 2709.196,E2 2709.196} C_VEL
LIN {X 0,Y 565.944,Z 656.68,A -85,B 0,C 180,E1 2709.919,E2 2709.919} C_VEL
LIN {X 0,Y 565.933,Z 655.527,A -85,B 0,C 180,E1 2710.012,E2 2710.012} C_VEL
LIN {X 0,Y 567.328,Z 619.286,A -85,B 0,C 180,E1 2712.489,E2 2712.489} C_VEL
LIN {X 0,Y 568.507,Z 580.557,A -85,B 0,C 180,E1 2714.376,E2 2714.376} C_VEL
LIN {X 0,Y 568.123,Z 565.186,A -85,B 0,C 180,E1 2714.978,E2 2714.978} C_VEL
LIN {X 0,Y 562.287,Z 549.53,A -85,B 0,C 180,E1 2715.91,E2 2715.91} C_VEL
LIN {X 0,Y 562.158,Z 549.53,A -85,B 0,C 180,E1 2722.148,E2 2722.148} C_VEL
LIN {X 0,Y 562.07,Z 549.53,A -85,B 0,C 180,E1 2727.259,E2 2727.259} C_VEL
LIN {X 0,Y 561.943,Z 549.53,A -85,B 0,C 180,E1 2732.602,E2 2732.602} C_VEL
LIN {X 0,Y 562.034,Z 549.53,A -85,B 0,C 180,E1 2738.281,E2 2738.281} C_VEL
LIN {X 0,Y 562.044,Z 549.53,A -85,B 0,C 180,E1 2744.453,E2 2744.453} C_VEL
LIN {X 0,Y 561.909,Z 549.53,A -85,B 0,C 180,E1 2749.707,E2 2749.707} C_VEL
LIN {X 0,Y 562.139,Z 549.53,A -85,B 0,C 180,E1 2755.554,E2 2755.554} C_VEL
LIN {X 0,Y 562.295,Z 550.037,A -85,B 0,C 180,E1 2757.747,E2 2757.747} C_VEL
LIN {X 0,Y 569.418,Z 566.255,A -85,B 0,C 180,E1 2758.434,E2 2758.434} C_VEL
LIN {X 0,Y 569.289,Z 624.54,A -85,B 0,C 180,E1 2759.422,E2 2759.422} C_VEL
LIN {X 0,Y 568.428,Z 663.282,A -85,B 0,C 180,E1 2760.687,E2 2760.687} C_VEL
LIN {X 0,Y 567.238,Z 701.236,A -85,B 0,C 180,E1 2762.581,E2 2762.581} C_VEL
LIN {X 0,Y 565.896,Z 736.696,A -85,B 0,C 180,E1 2765.042,E2 2765.042} C_VEL
LIN {X 0,Y 564.683,Z 768.227,A -85,B 0,C 180,E1 2767.952,E2 2767.952} C_VEL
LIN {X 0,Y 563.796,Z 795.23,A -85,B 0,C 180,E1 2771.2,E2 2771.2} C_VEL
LIN {X 0,Y 563.193,Z 817.455,A -85,B 0,C 180,E1 2774.693,E2 2774.693} C_VEL
LIN {X 0,Y 562.773,Z 834.823,A -85,B 0,C 180,E1 2778.358,E2 2778.358} C_VEL
LIN {X 0,Y 562.682,Z 847.611,A -85,B 0,C 180,E1 2782.267,E2 2782.267} C_VEL
LIN {X 0,Y 562.568,Z 853.931,A -85,B 0,C 180,E1 2785.368,E2 2785.368} C_VEL
LIN {X 0,Y 562.576,Z 857.083,A -85,B 0,C 180,E1 2788.457,E2 2788.457} C_VEL
LIN {X 0,Y 562.681,Z 857.084,A -85,B 0,C 180,E1 2791.541,E2 2791.541} C_VEL
LIN {X 0,Y 562.754,Z 852.531,A -85,B 0,C 180,E1 2795.506,E2 2795.506} C_VEL
LIN {X 0,Y 562.742,Z 841.962,A -85,B 0,C 180,E1 2799.68,E2 2799.68} C_VEL
LIN {X 0,Y 563.01,Z 826.222,A -85,B 0,C 180,E1 2803.609,E2 2803.609} C_VEL
LIN {X 0,Y 563.499,Z 806.285,A -85,B 0,C 180,E1 2807.19,E2 2807.19} C_VEL
LIN {X 0,Y 564.277,Z 781.006,A -85,B 0,C 180,E1 2810.619,E2 2810.619} C_VEL
LIN {X 0,Y 565.399,Z 750.404,A -85,B 0,C 180,E1 2813.787,E2 2813.787} C_VEL
LIN {X 0,Y 566.62,Z 716.922,A -85,B 0,C 180,E1 2816.421,E2 2816.421} C_VEL
LIN {X 0,Y 567.864,Z 682.217,A -85,B 0,C 180,E1 2818.45,E2 2818.45} C_VEL
LIN {X 0,Y 568.887,Z 646.508,A -85,B 0,C 180,E1 2819.931,E2 2819.931} C_VEL
LIN {X 0,Y 569.529,Z 608.118,A -85,B 0,C 180,E1 2820.926,E2 2820.926} C_VEL
LIN {X 0,Y 568.865,Z 565.478,A -85,B 0,C 180,E1 2821.612,E2 2821.612} C_VEL
LIN {X 0,Y 562.028,Z 549.53,A -85,B 0,C 180,E1 2822.321,E2 2822.321} C_VEL
LIN {X 0,Y 562.031,Z 549.53,A -85,B 0,C 180,E1 2828.286,E2 2828.286} C_VEL
LIN {X 0,Y 562.041,Z 549.53,A -85,B 0,C 180,E1 2834.459,E2 2834.459} C_VEL
LIN {X 0,Y 561.906,Z 549.53,A -85,B 0,C 180,E1 2839.713,E2 2839.713} C_VEL
LIN {X 0,Y 562.05,Z 549.53,A -85,B 0,C 180,E1 2845.554,E2 2845.554} C_VEL
LIN {X 0,Y 562.115,Z 549.53,A -85,B 0,C 180,E1 2851.003,E2 2851.003} C_VEL
LIN {X 0,Y 562.118,Z 549.53,A -85,B 0,C 180,E1 2856.317,E2 2856.317} C_VEL
LIN {X 0,Y 562.192,Z 549.53,A -85,B 0,C 180,E1 2861.149,E2 2861.149} C_VEL
LIN {X 0,Y 562.304,Z 549.53,A -85,B 0,C 180,E1 2867.564,E2 2867.564} C_VEL
LIN {X 0,Y 562.356,Z 549.53,A -85,B 0,C 180,E1 2872.267,E2 2872.267} C_VEL
LIN {X 0,Y 562.443,Z 549.53,A -85,B 0,C 180,E1 2876.917,E2 2876.917} C_VEL
LIN {X 0,Y 562.581,Z 549.53,A -85,B 0,C 180,E1 2881.545,E2 2881.545} C_VEL
LIN {X 0,Y 562.523,Z 549.53,A -85,B 0,C 180,E1 2886.184,E2 2886.184} C_VEL
LIN {X 0,Y 562.182,Z 549.53,A -85,B 0,C 180,E1 2892.445,E2 2892.445} C_VEL
LIN {X 0,Y 562.18,Z 549.53,A -85,B 0,C 180,E1 2897.236,E2 2897.236} C_VEL
LIN {X 0,Y 562.135,Z 549.53,A -85,B 0,C 180,E1 2902.156,E2 2902.156} C_VEL
LIN {X 0,Y 562.087,Z 549.53,A -85,B 0,C 180,E1 2907.266,E2 2907.266} C_VEL
LIN {X 0,Y 561.935,Z 549.53,A -85,B 0,C 180,E1 2912.61,E2 2912.61} C_VEL
LIN {X 0,Y 562.005,Z 549.53,A -85,B 0,C 180,E1 2918.292,E2 2918.292} C_VEL
LIN {X 0,Y 562.011,Z 549.53,A -85,B 0,C 180,E1 2924.466,E2 2924.466} C_VEL
LIN {X 0,Y 561.892,Z 549.53,A -85,B 0,C 180,E1 2929.708,E2 2929.708} C_VEL
LIN {X 0,Y 562.056,Z 549.53,A -85,B 0,C 180,E1 2935.55,E2 2935.55} C_VEL
LIN {X 0,Y 562.076,Z 549.53,A -85,B 0,C 180,E1 2940.997,E2 2940.997} C_VEL
LIN {X 0,Y 562.128,Z 549.53,A -85,B 0,C 180,E1 2946.32,E2 2946.32} C_VEL
LIN {X 0,Y 562.226,Z 549.53,A -85,B 0,C 180,E1 2951.147,E2 2951.147} C_VEL
LIN {X 0,Y 562.323,Z 549.53,A -85,B 0,C 180,E1 2957.562,E2 2957.562} C_VEL
LIN {X 0,Y 562.372,Z 549.53,A -85,B 0,C 180,E1 2962.264,E2 2962.264} C_VEL
LIN {X 0,Y 562.51,Z 549.53,A -85,B 0,C 180,E1 2966.915,E2 2966.915} C_VEL
LIN {X 0,Y 562.602,Z 549.53,A -85,B 0,C 180,E1 2971.543,E2 2971.543} C_VEL
LIN {X 0,Y 562.539,Z 549.53,A -85,B 0,C 180,E1 2976.181,E2 2976.181} C_VEL
LIN {X 0,Y 562.234,Z 549.53,A -85,B 0,C 180,E1 2982.442,E2 2982.442} C_VEL
LIN {X 0,Y 562.218,Z 549.53,A -85,B 0,C 180,E1 2987.232,E2 2987.232} C_VEL
LIN {X 0,Y 562.181,Z 549.53,A -85,B 0,C 180,E1 2992.152,E2 2992.152} C_VEL
LIN {X 0,Y 562.101,Z 549.53,A -85,B 0,C 180,E1 2997.263,E2 2997.263} C_VEL
LIN {X 0,Y 561.969,Z 549.53,A -85,B 0,C 180,E1 3002.606,E2 3002.606} C_VEL
LIN {X 0,Y 562.028,Z 549.53,A -85,B 0,C 180,E1 3008.288,E2 3008.288} C_VEL
LIN {X 0,Y 561.971,Z 549.966,A -85,B 0,C 180,E1 3014.086,E2 3014.086} C_VEL
LIN {X 0,Y 568.67,Z 569.194,A -85,B 0,C 180,E1 3015.103,E2 3015.103} C_VEL
LIN {X 0,Y 567.59,Z 608.569,A -85,B 0,C 180,E1 3016.821,E2 3016.821} C_VEL
LIN {X 0,Y 566.324,Z 645.372,A -85,B 0,C 180,E1 3019.125,E2 3019.125} C_VEL
LIN {X 0,Y 565.091,Z 678.825,A -85,B 0,C 180,E1 3021.955,E2 3021.955} C_VEL
LIN {X 0,Y 564.037,Z 708.069,A -85,B 0,C 180,E1 3025.206,E2 3025.206} C_VEL
LIN {X 0,Y 563.355,Z 733.071,A -85,B 0,C 180,E1 3028.869,E2 3028.869} C_VEL
LIN {X 0,Y 562.955,Z 752.724,A -85,B 0,C 180,E1 3032.79,E2 3032.79} C_VEL
LIN {X 0,Y 562.687,Z 766.019,A -85,B 0,C 180,E1 3036.613,E2 3036.613} C_VEL
LIN {X 0,Y 562.574,Z 774.046,A -85,B 0,C 180,E1 3040.386,E2 3040.386} C_VEL
LIN {X 0,Y 562.615,Z 777.397,A -85,B 0,C 180,E1 3044.386,E2 3044.386} C_VEL
LIN {X 0,Y 562.628,Z 776.38,A -85,B 0,C 180,E1 3047.565,E2 3047.565} C_VEL
LIN {X 0,Y 562.696,Z 770.48,A -85,B 0,C 180,E1 3051.486,E2 3051.486} C_VEL
LIN {X 0,Y 562.877,Z 759.457,A -85,B 0,C 180,E1 3055.368,E2 3055.368} C_VEL
LIN {X 0,Y 563.132,Z 742.941,A -85,B 0,C 180,E1 3059.227,E2 3059.227} C_VEL
LIN {X 0,Y 563.599,Z 721.397,A -85,B 0,C 180,E1 3062.884,E2 3062.884} C_VEL
LIN {X 0,Y 564.532,Z 694.593,A -85,B 0,C 180,E1 3066.316,E2 3066.316} C_VEL
LIN {X 0,Y 565.658,Z 662.559,A -85,B 0,C 180,E1 3069.432,E2 3069.432} C_VEL
LIN {X 0,Y 565.933,Z 655.527,A -85,B 0,C 180,E1 3070.012,E2 3070.012} C_VEL
LIN {X 0,Y 565.162,Z 648.834,A -85,B 0,C 180,E1 3070.579,E2 3070.579} C_VEL
LIN {X 0,Y 559.759,Z 630.919,A -85,B 0,C 180,E1 3072.147,E2 3072.147} C_VEL
LIN {X 0,Y 559.76,Z 629.075,A -85,B 0,C 180,E1 3072.269,E2 3072.269} C_VEL
LIN {X 0,Y 561.138,Z 591.593,A -85,B 0,C 180,E1 3074.309,E2 3074.309} C_VEL
LIN {X 0,Y 561.465,Z 568.512,A -85,B 0,C 180,E1 3075.256,E2 3075.256} C_VEL
LIN {X 0,Y 554.357,Z 549.53,A -85,B 0,C 180,E1 3076.373,E2 3076.373} C_VEL
LIN {X 0,Y 554.239,Z 549.53,A -85,B 0,C 180,E1 3082.481,E2 3082.481} C_VEL
LIN {X 0,Y 554.143,Z 549.53,A -85,B 0,C 180,E1 3087.672,E2 3087.672} C_VEL
LIN {X 0,Y 554.034,Z 549.53,A -85,B 0,C 180,E1 3093.126,E2 3093.126} C_VEL
LIN {X 0,Y 554.115,Z 549.53,A -85,B 0,C 180,E1 3098.931,E2 3098.931} C_VEL
LIN {X 0,Y 554.136,Z 549.53,A -85,B 0,C 180,E1 3104.732,E2 3104.732} C_VEL
LIN {X 0,Y 554.003,Z 549.53,A -85,B 0,C 180,E1 3111.054,E2 3111.054} C_VEL
LIN {X 0,Y 554.333,Z 549.53,A -85,B 0,C 180,E1 3117.202,E2 3117.202} C_VEL
LIN {X 0,Y 562.63,Z 568.743,A -85,B 0,C 180,E1 3118.045,E2 3118.045} C_VEL
LIN {X 0,Y 562.456,Z 625.162,A -85,B 0,C 180,E1 3119.028,E2 3119.028} C_VEL
LIN {X 0,Y 561.436,Z 664.273,A -85,B 0,C 180,E1 3120.331,E2 3120.331} C_VEL
LIN {X 0,Y 560.07,Z 701.196,A -85,B 0,C 180,E1 3122.197,E2 3122.197} C_VEL
LIN {X 0,Y 558.505,Z 737.115,A -85,B 0,C 180,E1 3124.724,E2 3124.724} C_VEL
LIN {X 0,Y 557.143,Z 768.226,A -85,B 0,C 180,E1 3127.637,E2 3127.637} C_VEL
LIN {X 0,Y 556.095,Z 795.232,A -85,B 0,C 180,E1 3130.929,E2 3130.929} C_VEL
LIN {X 0,Y 555.378,Z 817.266,A -85,B 0,C 180,E1 3134.437,E2 3134.437} C_VEL
LIN {X 0,Y 554.913,Z 834.824,A -85,B 0,C 180,E1 3138.191,E2 3138.191} C_VEL
LIN {X 0,Y 554.789,Z 847.612,A -85,B 0,C 180,E1 3142.157,E2 3142.157} C_VEL
LIN {X 0,Y 554.679,Z 853.931,A -85,B 0,C 180,E1 3145.302,E2 3145.302} C_VEL
LIN {X 0,Y 554.674,Z 857.083,A -85,B 0,C 180,E1 3148.435,E2 3148.435} C_VEL
LIN {X 0,Y 554.775,Z 857.084,A -85,B 0,C 180,E1 3151.563,E2 3151.563} C_VEL
LIN {X 0,Y 554.837,Z 852.531,A -85,B 0,C 180,E1 3155.585,E2 3155.585} C_VEL
LIN {X 0,Y 554.856,Z 842.105,A -85,B 0,C 180,E1 3159.776,E2 3159.776} C_VEL
LIN {X 0,Y 555.187,Z 826.22,A -85,B 0,C 180,E1 3163.805,E2 3163.805} C_VEL
LIN {X 0,Y 555.741,Z 805.565,A -85,B 0,C 180,E1 3167.549,E2 3167.549} C_VEL
LIN {X 0,Y 556.758,Z 779.253,A -85,B 0,C 180,E1 3171.119,E2 3171.119} C_VEL
LIN {X 0,Y 558.002,Z 749.777,A -85,B 0,C 180,E1 3174.18,E2 3174.18} C_VEL
LIN {X 0,Y 559.42,Z 716.261,A -85,B 0,C 180,E1 3176.835,E2 3176.835} C_VEL
LIN {X 0,Y 560.839,Z 680.742,A -85,B 0,C 180,E1 3178.916,E2 3178.916} C_VEL
LIN {X 0,Y 562.058,Z 644.455,A -85,B 0,C 180,E1 3180.403,E2 3180.403} C_VEL
LIN {X 0,Y 562.766,Z 606.364,A -85,B 0,C 180,E1 3181.369,E2 3181.369} C_VEL
LIN {X 0,Y 562.119,Z 567.853,A -85,B 0,C 180,E1 3182.001,E2 3182.001} C_VEL
LIN {X 0,Y 554.057,Z 549.53,A -85,B 0,C 180,E1 3182.865,E2 3182.865} C_VEL
LIN {X 0,Y 554.116,Z 549.53,A -85,B 0,C 180,E1 3188.935,E2 3188.935} C_VEL
LIN {X 0,Y 554.131,Z 549.53,A -85,B 0,C 180,E1 3194.738,E2 3194.738} C_VEL
LIN {X 0,Y 553.996,Z 549.53,A -85,B 0,C 180,E1 3201.059,E2 3201.059} C_VEL
LIN {X 0,Y 554.212,Z 549.53,A -85,B 0,C 180,E1 3206.886,E2 3206.886} C_VEL
LIN {X 0,Y 554.154,Z 549.53,A -85,B 0,C 180,E1 3212.328,E2 3212.328} C_VEL
LIN {X 0,Y 554.133,Z 549.53,A -85,B 0,C 180,E1 3218.275,E2 3218.275} C_VEL
LIN {X 0,Y 554.315,Z 549.53,A -85,B 0,C 180,E1 3222.937,E2 3222.937} C_VEL
LIN {X 0,Y 554.382,Z 549.53,A -85,B 0,C 180,E1 3227.384,E2 3227.384} C_VEL
LIN {X 0,Y 554.443,Z 549.53,A -85,B 0,C 180,E1 3232.156,E2 3232.156} C_VEL
LIN {X 0,Y 554.557,Z 549.53,A -85,B 0,C 180,E1 3236.873,E2 3236.873} C_VEL
LIN {X 0,Y 554.671,Z 549.53,A -85,B 0,C 180,E1 3241.567,E2 3241.567} C_VEL
LIN {X 0,Y 554.592,Z 549.53,A -85,B 0,C 180,E1 3246.272,E2 3246.272} C_VEL
LIN {X 0,Y 554.264,Z 549.53,A -85,B 0,C 180,E1 3252.626,E2 3252.626} C_VEL
LIN {X 0,Y 554.263,Z 549.53,A -85,B 0,C 180,E1 3257.49,E2 3257.49} C_VEL
LIN {X 0,Y 554.219,Z 549.53,A -85,B 0,C 180,E1 3262.489,E2 3262.489} C_VEL
LIN {X 0,Y 554.151,Z 549.53,A -85,B 0,C 180,E1 3267.679,E2 3267.679} C_VEL
LIN {X 0,Y 554.035,Z 549.53,A -85,B 0,C 180,E1 3273.134,E2 3273.134} C_VEL
LIN {X 0,Y 554.064,Z 549.53,A -85,B 0,C 180,E1 3278.943,E2 3278.943} C_VEL
LIN {X 0,Y 554.112,Z 549.53,A -85,B 0,C 180,E1 3284.731,E2 3284.731} C_VEL
LIN {X 0,Y 553.972,Z 549.53,A -85,B 0,C 180,E1 3289.934,E2 3289.934} C_VEL
LIN {X 0,Y 554.109,Z 549.53,A -85,B 0,C 180,E1 3295.061,E2 3295.061} C_VEL
LIN {X 0,Y 554.194,Z 549.53,A -85,B 0,C 180,E1 3300.96,E2 3300.96} C_VEL
LIN {X 0,Y 554.14,Z 549.53,A -85,B 0,C 180,E1 3305.806,E2 3305.806} C_VEL
LIN {X 0,Y 554.281,Z 549.53,A -85,B 0,C 180,E1 3310.866,E2 3310.866} C_VEL
LIN {X 0,Y 554.412,Z 549.53,A -85,B 0,C 180,E1 3315.772,E2 3315.772} C_VEL
LIN {X 0,Y 554.457,Z 549.53,A -85,B 0,C 180,E1 3322.153,E2 3322.153} C_VEL
LIN {X 0,Y 554.622,Z 549.53,A -85,B 0,C 180,E1 3326.871,E2 3326.871} C_VEL
LIN {X 0,Y 554.691,Z 549.53,A -85,B 0,C 180,E1 3331.565,E2 3331.565} C_VEL
LIN {X 0,Y 554.609,Z 549.53,A -85,B 0,C 180,E1 3336.27,E2 3336.27} C_VEL
LIN {X 0,Y 554.313,Z 549.53,A -85,B 0,C 180,E1 3342.622,E2 3342.622} C_VEL
LIN {X 0,Y 554.295,Z 549.53,A -85,B 0,C 180,E1 3347.486,E2 3347.486} C_VEL
LIN {X 0,Y 554.264,Z 549.53,A -85,B 0,C 180,E1 3352.485,E2 3352.485} C_VEL
LIN {X 0,Y 554.172,Z 549.53,A -85,B 0,C 180,E1 3357.676,E2 3357.676} C_VEL
LIN {X 0,Y 554.063,Z 549.53,A -85,B 0,C 180,E1 3363.13,E2 3363.13} C_VEL
LIN {X 0,Y 554.075,Z 549.53,A -85,B 0,C 180,E1 3368.94,E2 3368.94} C_VEL
LIN {X 0,Y 554.04,Z 549.775,A -85,B 0,C 180,E1 3373.589,E2 3373.589} C_VEL
LIN {X 0,Y 561.717,Z 571.667,A -85,B 0,C 180,E1 3374.787,E2 3374.787} C_VEL
LIN {X 0,Y 560.453,Z 611.035,A -85,B 0,C 180,E1 3376.569,E2 3376.569} C_VEL
LIN {X 0,Y 558.924,Z 647.746,A -85,B 0,C 180,E1 3378.942,E2 3378.942} C_VEL
LIN {X 0,Y 557.503,Z 680.998,A -85,B 0,C 180,E1 3381.843,E2 3381.843} C_VEL
LIN {X 0,Y 556.344,Z 709.78,A -85,B 0,C 180,E1 3385.142,E2 3385.142} C_VEL
LIN {X 0,Y 555.548,Z 734.797,A -85,B 0,C 180,E1 3388.94,E2 3388.94} C_VEL
LIN {X 0,Y 555.105,Z 753.524,A -85,B 0,C 180,E1 3392.812,E2 3392.812} C_VEL
LIN {X 0,Y 554.804,Z 766.635,A -85,B 0,C 180,E1 3396.717,E2 3396.717} C_VEL
LIN {X 0,Y 554.652,Z 774.857,A -85,B 0,C 180,E1 3400.876,E2 3400.876} C_VEL
LIN {X 0,Y 554.679,Z 777.352,A -85,B 0,C 180,E1 3404.156,E2 3404.156} C_VEL
LIN {X 0,Y 554.704,Z 776.542,A -85,B 0,C 180,E1 3407.384,E2 3407.384} C_VEL
LIN {X 0,Y 554.776,Z 770.909,A -85,B 0,C 180,E1 3411.364,E2 3411.364} C_VEL
LIN {X 0,Y 554.994,Z 760.189,A -85,B 0,C 180,E1 3415.302,E2 3415.302} C_VEL
LIN {X 0,Y 555.27,Z 744.003,A -85,B 0,C 180,E1 3419.216,E2 3419.216} C_VEL
LIN {X 0,Y 555.835,Z 722.828,A -85,B 0,C 180,E1 3422.924,E2 3422.924} C_VEL
LIN {X 0,Y 556.902,Z 696.477,A -85,B 0,C 180,E1 3426.403,E2 3426.403} C_VEL
LIN {X 0,Y 558.22,Z 665.105,A -85,B 0,C 180,E1 3429.559,E2 3429.559} C_VEL
LIN {X 0,Y 559.76,Z 629.075,A -85,B 0,C 180,E1 3432.269,E2 3432.269} C_VEL
LIN {X 0,Y 556.742,Z 615.049,A -85,B 0,C 180,E1 3433.312,E2 3433.312} C_VEL
LIN {X 0,Y 553.826,Z 601.566,A -85,B 0,C 180,E1 3434.231,E2 3434.231} C_VEL
LIN {X 0,Y 553.865,Z 600.585,A -85,B 0,C 180,E1 3434.281,E2 3434.281} C_VEL
LIN {X 0,Y 554.44,Z 570.701,A -85,B 0,C 180,E1 3435.598,E2 3435.598} C_VEL
LIN {X 0,Y 546.42,Z 549.53,A -85,B 0,C 180,E1 3436.886,E2 3436.886} C_VEL
LIN {X 0,Y 546.297,Z 549.53,A -85,B 0,C 180,E1 3442.827,E2 3442.827} C_VEL
LIN {X 0,Y 546.218,Z 549.53,A -85,B 0,C 180,E1 3448.109,E2 3448.109} C_VEL
LIN {X 0,Y 546.113,Z 549.53,A -85,B 0,C 180,E1 3453.722,E2 3453.722} C_VEL
LIN {X 0,Y 546.187,Z 549.53,A -85,B 0,C 180,E1 3459.606,E2 3459.606} C_VEL
LIN {X 0,Y 546.19,Z 549.53,A -85,B 0,C 180,E1 3463.884,E2 3463.884} C_VEL
LIN {X 0,Y 546.086,Z 549.53,A -85,B 0,C 180,E1 3470.379,E2 3470.379} C_VEL
LIN {X 0,Y 546.385,Z 550.239,A -85,B 0,C 180,E1 3476.691,E2 3476.691} C_VEL
LIN {X 0,Y 556.067,Z 572.92,A -85,B 0,C 180,E1 3477.684,E2 3477.684} C_VEL
LIN {X 0,Y 555.65,Z 625.519,A -85,B 0,C 180,E1 3478.616,E2 3478.616} C_VEL
LIN {X 0,Y 554.57,Z 663.493,A -85,B 0,C 180,E1 3479.89,E2 3479.89} C_VEL
LIN {X 0,Y 552.988,Z 701.231,A -85,B 0,C 180,E1 3481.812,E2 3481.812} C_VEL
LIN {X 0,Y 551.182,Z 737.054,A -85,B 0,C 180,E1 3484.359,E2 3484.359} C_VEL
LIN {X 0,Y 549.616,Z 768.226,A -85,B 0,C 180,E1 3487.314,E2 3487.314} C_VEL
LIN {X 0,Y 548.398,Z 795.233,A -85,B 0,C 180,E1 3490.651,E2 3490.651} C_VEL
LIN {X 0,Y 547.573,Z 816.963,A -85,B 0,C 180,E1 3494.152,E2 3494.152} C_VEL
LIN {X 0,Y 547.042,Z 834.824,A -85,B 0,C 180,E1 3498.019,E2 3498.019} C_VEL
LIN {X 0,Y 546.955,Z 846.644,A -85,B 0,C 180,E1 3501.643,E2 3501.643} C_VEL
LIN {X 0,Y 546.786,Z 854.165,A -85,B 0,C 180,E1 3505.389,E2 3505.389} C_VEL
LIN {X 0,Y 546.772,Z 857.083,A -85,B 0,C 180,E1 3508.413,E2 3508.413} C_VEL
LIN {X 0,Y 546.869,Z 857.084,A -85,B 0,C 180,E1 3511.586,E2 3511.586} C_VEL
LIN {X 0,Y 546.939,Z 852.851,A -85,B 0,C 180,E1 3515.48,E2 3515.48} C_VEL
LIN {X 0,Y 547.002,Z 843.213,A -85,B 0,C 180,E1 3519.559,E2 3519.559} C_VEL
LIN {X 0,Y 547.35,Z 828.087,A -85,B 0,C 180,E1 3523.598,E2 3523.598} C_VEL
LIN {X 0,Y 547.959,Z 807.628,A -85,B 0,C 180,E1 3527.477,E2 3527.477} C_VEL
LIN {X 0,Y 549.115,Z 781.004,A -85,B 0,C 180,E1 3531.216,E2 3531.216} C_VEL
LIN {X 0,Y 550.524,Z 751.542,A -85,B 0,C 180,E1 3534.363,E2 3534.363} C_VEL
LIN {X 0,Y 552.065,Z 719.348,A -85,B 0,C 180,E1 3536.998,E2 3536.998} C_VEL
LIN {X 0,Y 553.715,Z 683.946,A -85,B 0,C 180,E1 3539.155,E2 3539.155} C_VEL
LIN {X 0,Y 555.157,Z 646.531,A -85,B 0,C 180,E1 3540.749,E2 3540.749} C_VEL
LIN {X 0,Y 556.028,Z 607.699,A -85,B 0,C 180,E1 3541.77,E2 3541.77} C_VEL
LIN {X 0,Y 555.416,Z 570.506,A -85,B 0,C 180,E1 3542.394,E2 3542.394} C_VEL
LIN {X 0,Y 546.134,Z 549.53,A -85,B 0,C 180,E1 3543.386,E2 3543.386} C_VEL
LIN {X 0,Y 546.191,Z 549.53,A -85,B 0,C 180,E1 3549.61,E2 3549.61} C_VEL
LIN {X 0,Y 546.185,Z 549.53,A -85,B 0,C 180,E1 3553.891,E2 3553.891} C_VEL
LIN {X 0,Y 546.081,Z 549.53,A -85,B 0,C 180,E1 3560.385,E2 3560.385} C_VEL
LIN {X 0,Y 546.216,Z 549.53,A -85,B 0,C 180,E1 3566.337,E2 3566.337} C_VEL
LIN {X 0,Y 546.254,Z 549.53,A -85,B 0,C 180,E1 3572.491,E2 3572.491} C_VEL
LIN {X 0,Y 546.208,Z 549.53,A -85,B 0,C 180,E1 3577.17,E2 3577.17} C_VEL
LIN {X 0,Y 546.371,Z 549.53,A -85,B 0,C 180,E1 3582.256,E2 3582.256} C_VEL
LIN {X 0,Y 546.458,Z 549.53,A -85,B 0,C 180,E1 3587.198,E2 3587.198} C_VEL
LIN {X 0,Y 546.527,Z 549.53,A -85,B 0,C 180,E1 3592.042,E2 3592.042} C_VEL
LIN {X 0,Y 546.647,Z 549.53,A -85,B 0,C 180,E1 3596.828,E2 3596.828} C_VEL
LIN {X 0,Y 546.762,Z 549.53,A -85,B 0,C 180,E1 3601.59,E2 3601.59} C_VEL
LIN {X 0,Y 546.686,Z 549.53,A -85,B 0,C 180,E1 3606.364,E2 3606.364} C_VEL
LIN {X 0,Y 546.349,Z 549.53,A -85,B 0,C 180,E1 3612.812,E2 3612.812} C_VEL
LIN {X 0,Y 546.331,Z 549.53,A -85,B 0,C 180,E1 3617.752,E2 3617.752} C_VEL
LIN {X 0,Y 546.28,Z 549.53,A -85,B 0,C 180,E1 3622.835,E2 3622.835} C_VEL
LIN {X 0,Y 546.22,Z 549.53,A -85,B 0,C 180,E1 3628.117,E2 3628.117} C_VEL
LIN {X 0,Y 546.085,Z 549.53,A -85,B 0,C 180,E1 3633.72,E2 3633.72} C_VEL
LIN {X 0,Y 546.146,Z 549.53,A -85,B 0,C 180,E1 3639.618,E2 3639.618} C_VEL
LIN {X 0,Y 546.174,Z 549.53,A -85,B 0,C 180,E1 3643.884,E2 3643.884} C_VEL
LIN {X 0,Y 546.075,Z 549.53,A -85,B 0,C 180,E1 3650.38,E2 3650.38} C_VEL
LIN {X 0,Y 546.226,Z 549.53,A -85,B 0,C 180,E1 3656.333,E2 3656.333} C_VEL
LIN {X 0,Y 546.198,Z 549.53,A -85,B 0,C 180,E1 3661.886,E2 3661.886} C_VEL
LIN {X 0,Y 546.222,Z 549.53,A -85,B 0,C 180,E1 3667.167,E2 3667.167} C_VEL
LIN {X 0,Y 546.404,Z 549.53,A -85,B 0,C 180,E1 3672.254,E2 3672.254} C_VEL
LIN {X 0,Y 546.48,Z 549.53,A -85,B 0,C 180,E1 3677.195,E2 3677.195} C_VEL
LIN {X 0,Y 546.541,Z 549.53,A -85,B 0,C 180,E1 3682.039,E2 3682.039} C_VEL
LIN {X 0,Y 546.712,Z 549.53,A -85,B 0,C 180,E1 3686.826,E2 3686.826} C_VEL
LIN {X 0,Y 546.782,Z 549.53,A -85,B 0,C 180,E1 3691.587,E2 3691.587} C_VEL
LIN {X 0,Y 546.704,Z 549.53,A -85,B 0,C 180,E1 3696.361,E2 3696.361} C_VEL
LIN {X 0,Y 546.394,Z 549.53,A -85,B 0,C 180,E1 3702.809,E2 3702.809} C_VEL
LIN {X 0,Y 546.36,Z 549.53,A -85,B 0,C 180,E1 3707.749,E2 3707.749} C_VEL
LIN {X 0,Y 546.326,Z 549.53,A -85,B 0,C 180,E1 3712.83,E2 3712.83} C_VEL
LIN {X 0,Y 546.246,Z 549.53,A -85,B 0,C 180,E1 3718.113,E2 3718.113} C_VEL
LIN {X 0,Y 546.121,Z 549.53,A -85,B 0,C 180,E1 3723.721,E2 3723.721} C_VEL
LIN {X 0,Y 546.142,Z 549.53,A -85,B 0,C 180,E1 3729.616,E2 3729.616} C_VEL
LIN {X 0,Y 546.113,Z 549.53,A -85,B 0,C 180,E1 3733.062,E2 3733.062} C_VEL
LIN {X 0,Y 554.773,Z 573.642,A -85,B 0,C 180,E1 3734.448,E2 3734.448} C_VEL
LIN {X 0,Y 553.32,Z 612.72,A -85,B 0,C 180,E1 3736.269,E2 3736.269} C_VEL
LIN {X 0,Y 551.633,Z 648.414,A -85,B 0,C 180,E1 3738.625,E2 3738.625} C_VEL
LIN {X 0,Y 550.052,Z 680.726,A -85,B 0,C 180,E1 3741.483,E2 3741.483} C_VEL
LIN {X 0,Y 548.648,Z 710.508,A -85,B 0,C 180,E1 3744.948,E2 3744.948} C_VEL
LIN {X 0,Y 547.733,Z 734.702,A -85,B 0,C 180,E1 3748.688,E2 3748.688} C_VEL
LIN {X 0,Y 547.267,Z 753.589,A -85,B 0,C 180,E1 3752.652,E2 3752.652} C_VEL
LIN {X 0,Y 546.915,Z 766.613,A -85,B 0,C 180,E1 3756.589,E2 3756.589} C_VEL
LIN {X 0,Y 546.749,Z 774.548,A -85,B 0,C 180,E1 3760.588,E2 3760.588} C_VEL
LIN {X 0,Y 546.759,Z 777.307,A -85,B 0,C 180,E1 3763.921,E2 3763.921} C_VEL
LIN {X 0,Y 546.781,Z 776.685,A -85,B 0,C 180,E1 3767.198,E2 3767.198} C_VEL
LIN {X 0,Y 546.868,Z 771.254,A -85,B 0,C 180,E1 3771.28,E2 3771.28} C_VEL
LIN {X 0,Y 547.108,Z 760.921,A -85,B 0,C 180,E1 3775.235,E2 3775.235} C_VEL
LIN {X 0,Y 547.419,Z 745.064,A -85,B 0,C 180,E1 3779.204,E2 3779.204} C_VEL
LIN {X 0,Y 548.063,Z 724.261,A -85,B 0,C 180,E1 3782.966,E2 3782.966} C_VEL
LIN {X 0,Y 549.237,Z 698.104,A -85,B 0,C 180,E1 3786.521,E2 3786.521} C_VEL
LIN {X 0,Y 550.768,Z 666.443,A -85,B 0,C 180,E1 3789.79,E2 3789.79} C_VEL
LIN {X 0,Y 552.448,Z 632.024,A -85,B 0,C 180,E1 3792.46,E2 3792.46} C_VEL
LIN {X 0,Y 553.865,Z 600.585,A -85,B 0,C 180,E1 3794.281,E2 3794.281} C_VEL
LIN {X 0,Y 551.899,Z 585.297,A -85,B 0,C 180,E1 3795.147,E2 3795.147} C_VEL
LIN {X 0,Y 546.541,Z 570.86,A -85,B 0,C 180,E1 3796.083,E2 3796.083} C_VEL
LIN {X 0,Y 538.483,Z 549.53,A -85,B 0,C 180,E1 3797.367,E2 3797.367} C_VEL
LIN {X 0,Y 538.386,Z 549.53,A -85,B 0,C 180,E1 3803.181,E2 3803.181} C_VEL
LIN {X 0,Y 538.248,Z 549.53,A -85,B 0,C 180,E1 3808.563,E2 3808.563} C_VEL
LIN {X 0,Y 538.175,Z 549.53,A -85,B 0,C 180,E1 3814.235,E2 3814.235} C_VEL
LIN {X 0,Y 538.212,Z 549.53,A -85,B 0,C 180,E1 3820.312,E2 3820.312} C_VEL
LIN {X 0,Y 538.19,Z 549.53,A -85,B 0,C 180,E1 3825.306,E2 3825.306} C_VEL
LIN {X 0,Y 538.185,Z 549.53,A -85,B 0,C 180,E1 3831.965,E2 3831.965} C_VEL
LIN {X 0,Y 538.368,Z 549.53,A -85,B 0,C 180,E1 3836.095,E2 3836.095} C_VEL
LIN {X 0,Y 549.39,Z 573.955,A -85,B 0,C 180,E1 3837.259,E2 3837.259} C_VEL
LIN {X 0,Y 548.883,Z 625.517,A -85,B 0,C 180,E1 3838.184,E2 3838.184} C_VEL
LIN {X 0,Y 547.617,Z 664.394,A -85,B 0,C 180,E1 3839.51,E2 3839.51} C_VEL
LIN {X 0,Y 545.911,Z 700.717,A -85,B 0,C 180,E1 3841.379,E2 3841.379} C_VEL
LIN {X 0,Y 543.985,Z 735.497,A -85,B 0,C 180,E1 3843.858,E2 3843.858} C_VEL
LIN {X 0,Y 542.275,Z 766.307,A -85,B 0,C 180,E1 3846.772,E2 3846.772} C_VEL
LIN {X 0,Y 540.797,Z 793.867,A -85,B 0,C 180,E1 3850.17,E2 3850.17} C_VEL
LIN {X 0,Y 539.774,Z 816.972,A -85,B 0,C 180,E1 3853.918,E2 3853.918} C_VEL
LIN {X 0,Y 539.187,Z 834.825,A -85,B 0,C 180,E1 3857.842,E2 3857.842} C_VEL
LIN {X 0,Y 539.054,Z 846.644,A -85,B 0,C 180,E1 3861.52,E2 3861.52} C_VEL
LIN {X 0,Y 538.887,Z 853.932,A -85,B 0,C 180,E1 3865.164,E2 3865.164} C_VEL
LIN {X 0,Y 538.887,Z 857.083,A -85,B 0,C 180,E1 3868.389,E2 3868.389} C_VEL
LIN {X 0,Y 538.977,Z 857.085,A -85,B 0,C 180,E1 3871.609,E2 3871.609} C_VEL
LIN {X 0,Y 539.015,Z 852.726,A -85,B 0,C 180,E1 3875.641,E2 3875.641} C_VEL
LIN {X 0,Y 539.097,Z 843.213,A -85,B 0,C 180,E1 3879.701,E2 3879.701} C_VEL
LIN {X 0,Y 539.498,Z 828.131,A -85,B 0,C 180,E1 3883.79,E2 3883.79} C_VEL
LIN {X 0,Y 540.202,Z 808.052,A -85,B 0,C 180,E1 3887.663,E2 3887.663} C_VEL
LIN {X 0,Y 541.53,Z 781.187,A -85,B 0,C 180,E1 3891.505,E2 3891.505} C_VEL
LIN {X 0,Y 543.082,Z 751.544,A -85,B 0,C 180,E1 3894.719,E2 3894.719} C_VEL
LIN {X 0,Y 544.955,Z 717.873,A -85,B 0,C 180,E1 3897.488,E2 3897.488} C_VEL
LIN {X 0,Y 546.821,Z 681.628,A -85,B 0,C 180,E1 3899.683,E2 3899.683} C_VEL
LIN {X 0,Y 548.338,Z 645.612,A -85,B 0,C 180,E1 3901.207,E2 3901.207} C_VEL
LIN {X 0,Y 549.311,Z 607.994,A -85,B 0,C 180,E1 3902.2,E2 3902.2} C_VEL
LIN {X 0,Y 548.861,Z 573.324,A -85,B 0,C 180,E1 3902.786,E2 3902.786} C_VEL
LIN {X 0,Y 538.185,Z 549.53,A -85,B 0,C 180,E1 3903.946,E2 3903.946} C_VEL
LIN {X 0,Y 538.276,Z 549.53,A -85,B 0,C 180,E1 3908.229,E2 3908.229} C_VEL
LIN {X 0,Y 538.196,Z 549.53,A -85,B 0,C 180,E1 3914.692,E2 3914.692} C_VEL
LIN {X 0,Y 538.116,Z 549.53,A -85,B 0,C 180,E1 3919.68,E2 3919.68} C_VEL
LIN {X 0,Y 538.237,Z 549.53,A -85,B 0,C 180,E1 3925.769,E2 3925.769} C_VEL
LIN {X 0,Y 538.296,Z 549.53,A -85,B 0,C 180,E1 3931.439,E2 3931.439} C_VEL
LIN {X 0,Y 538.305,Z 549.53,A -85,B 0,C 180,E1 3936.815,E2 3936.815} C_VEL
LIN {X 0,Y 538.419,Z 549.53,A -85,B 0,C 180,E1 3942.957,E2 3942.957} C_VEL
LIN {X 0,Y 538.515,Z 549.53,A -85,B 0,C 180,E1 3948.653,E2 3948.653} C_VEL
LIN {X 0,Y 538.572,Z 549.53,A -85,B 0,C 180,E1 3953.547,E2 3953.547} C_VEL
LIN {X 0,Y 538.619,Z 549.53,A -85,B 0,C 180,E1 3958.393,E2 3958.393} C_VEL
LIN {X 0,Y 538.618,Z 549.53,A -85,B 0,C 180,E1 3963.226,E2 3963.226} C_VEL
LIN {X 0,Y 538.5,Z 549.53,A -85,B 0,C 180,E1 3968.085,E2 3968.085} C_VEL
LIN {X 0,Y 538.46,Z 549.53,A -85,B 0,C 180,E1 3973.003,E2 3973.003} C_VEL
LIN {X 0,Y 538.427,Z 549.53,A -85,B 0,C 180,E1 3978.021,E2 3978.021} C_VEL
LIN {X 0,Y 538.376,Z 549.53,A -85,B 0,C 180,E1 3983.189,E2 3983.189} C_VEL
LIN {X 0,Y 538.247,Z 549.53,A -85,B 0,C 180,E1 3988.571,E2 3988.571} C_VEL
LIN {X 0,Y 538.154,Z 549.53,A -85,B 0,C 180,E1 3994.245,E2 3994.245} C_VEL
LIN {X 0,Y 538.182,Z 549.53,A -85,B 0,C 180,E1 4000.323,E2 4000.323} C_VEL
LIN {X 0,Y 538.147,Z 549.53,A -85,B 0,C 180,E1 4005.303,E2 4005.303} C_VEL
LIN {X 0,Y 538.174,Z 549.53,A -85,B 0,C 180,E1 4011.763,E2 4011.763} C_VEL
LIN {X 0,Y 538.293,Z 549.53,A -85,B 0,C 180,E1 4017.697,E2 4017.697} C_VEL
LIN {X 0,Y 538.237,Z 549.53,A -85,B 0,C 180,E1 4023.252,E2 4023.252} C_VEL
LIN {X 0,Y 538.317,Z 549.53,A -85,B 0,C 180,E1 4028.554,E2 4028.554} C_VEL
LIN {X 0,Y 538.433,Z 549.53,A -85,B 0,C 180,E1 4033.669,E2 4033.669} C_VEL
LIN {X 0,Y 538.524,Z 549.53,A -85,B 0,C 180,E1 4038.65,E2 4038.65} C_VEL
LIN {X 0,Y 538.597,Z 549.53,A -85,B 0,C 180,E1 4043.544,E2 4043.544} C_VEL
LIN {X 0,Y 538.668,Z 549.53,A -85,B 0,C 180,E1 4048.39,E2 4048.39} C_VEL
LIN {X 0,Y 538.631,Z 549.53,A -85,B 0,C 180,E1 4053.224,E2 4053.224} C_VEL
LIN {X 0,Y 538.522,Z 549.53,A -85,B 0,C 180,E1 4058.082,E2 4058.082} C_VEL
LIN {X 0,Y 538.499,Z 549.53,A -85,B 0,C 180,E1 4063,E2 4063} C_VEL
LIN {X 0,Y 538.454,Z 549.53,A -85,B 0,C 180,E1 4068.018,E2 4068.018} C_VEL
LIN {X 0,Y 538.419,Z 549.53,A -85,B 0,C 180,E1 4073.185,E2 4073.185} C_VEL
LIN {X 0,Y 538.276,Z 549.53,A -85,B 0,C 180,E1 4078.567,E2 4078.567} C_VEL
LIN {X 0,Y 538.189,Z 549.53,A -85,B 0,C 180,E1 4084.24,E2 4084.24} C_VEL
LIN {X 0,Y 538.167,Z 549.53,A -85,B 0,C 180,E1 4090.322,E2 4090.322} C_VEL
LIN {X 0,Y 538.248,Z 549.53,A -85,B 0,C 180,E1 4092.522,E2 4092.522} C_VEL
LIN {X 0,Y 547.809,Z 576.388,A -85,B 0,C 180,E1 4094.131,E2 4094.131} C_VEL
LIN {X 0,Y 546.211,Z 614.15,A -85,B 0,C 180,E1 4095.946,E2 4095.946} C_VEL
LIN {X 0,Y 544.282,Z 650.409,A -85,B 0,C 180,E1 4098.402,E2 4098.402} C_VEL
LIN {X 0,Y 542.453,Z 683.263,A -85,B 0,C 180,E1 4101.401,E2 4101.401} C_VEL
LIN {X 0,Y 540.91,Z 712.628,A -85,B 0,C 180,E1 4104.949,E2 4104.949} C_VEL
LIN {X 0,Y 539.916,Z 736.804,A -85,B 0,C 180,E1 4108.842,E2 4108.842} C_VEL
LIN {X 0,Y 539.328,Z 755.452,A -85,B 0,C 180,E1 4112.962,E2 4112.962} C_VEL
LIN {X 0,Y 538.998,Z 767.543,A -85,B 0,C 180,E1 4116.839,E2 4116.839} C_VEL
LIN {X 0,Y 538.859,Z 774.216,A -85,B 0,C 180,E1 4120.292,E2 4120.292} C_VEL
LIN {X 0,Y 538.825,Z 777.249,A -85,B 0,C 180,E1 4123.677,E2 4123.677} C_VEL
LIN {X 0,Y 538.895,Z 776.828,A -85,B 0,C 180,E1 4127.008,E2 4127.008} C_VEL
LIN {X 0,Y 538.96,Z 771.431,A -85,B 0,C 180,E1 4131.283,E2 4131.283} C_VEL
LIN {X 0,Y 539.225,Z 761.652,A -85,B 0,C 180,E1 4135.165,E2 4135.165} C_VEL
LIN {X 0,Y 539.584,Z 746.123,A -85,B 0,C 180,E1 4139.193,E2 4139.193} C_VEL
LIN {X 0,Y 540.327,Z 724.413,A -85,B 0,C 180,E1 4143.209,E2 4143.209} C_VEL
LIN {X 0,Y 541.674,Z 698.249,A -85,B 0,C 180,E1 4146.82,E2 4146.82} C_VEL
LIN {X 0,Y 543.364,Z 666.7,A -85,B 0,C 180,E1 4150.127,E2 4150.127} C_VEL
LIN {X 0,Y 545.303,Z 632.332,A -85,B 0,C 180,E1 4152.83,E2 4152.83} C_VEL
LIN {X 0,Y 547.132,Z 594.614,A -85,B 0,C 180,E1 4154.989,E2 4154.989} C_VEL
LIN {X 0,Y 547.486,Z 573.362,A -85,B 0,C 180,E1 4155.926,E2 4155.926} C_VEL
LIN {X 0,Y 546.541,Z 570.86,A -85,B 0,C 180,E1 4156.083,E2 4156.083} C_VEL
LIN {X 0,Y 539.732,Z 563.847,A -85,B 0,C 180,E1 4156.794,E2 4156.794} C_VEL
LIN {X 0,Y 532.957,Z 556.696,A -85,B 0,C 180,E1 4157.494,E2 4157.494} C_VEL
LIN {X 0,Y 530.549,Z 549.53,A -85,B 0,C 180,E1 4157.901,E2 4157.901} C_VEL
LIN {X 0,Y 530.438,Z 549.53,A -85,B 0,C 180,E1 4164.019,E2 4164.019} C_VEL
LIN {X 0,Y 530.331,Z 549.53,A -85,B 0,C 180,E1 4169.03,E2 4169.03} C_VEL
LIN {X 0,Y 530.271,Z 549.53,A -85,B 0,C 180,E1 4174.818,E2 4174.818} C_VEL
LIN {X 0,Y 530.279,Z 549.53,A -85,B 0,C 180,E1 4181.043,E2 4181.043} C_VEL
LIN {X 0,Y 530.262,Z 549.53,A -85,B 0,C 180,E1 4186.742,E2 4186.742} C_VEL
LIN {X 0,Y 530.233,Z 549.53,A -85,B 0,C 180,E1 4193.154,E2 4193.154} C_VEL
LIN {X 0,Y 530.388,Z 549.579,A -85,B 0,C 180,E1 4195.537,E2 4195.537} C_VEL
LIN {X 0,Y 542.594,Z 576.112,A -85,B 0,C 180,E1 4196.829,E2 4196.829} C_VEL
LIN {X 0,Y 542.106,Z 626.936,A -85,B 0,C 180,E1 4197.781,E2 4197.781} C_VEL
LIN {X 0,Y 540.708,Z 664.562,A -85,B 0,C 180,E1 4199.086,E2 4199.086} C_VEL
LIN {X 0,Y 538.821,Z 700.835,A -85,B 0,C 180,E1 4200.975,E2 4200.975} C_VEL
LIN {X 0,Y 536.666,Z 735.752,A -85,B 0,C 180,E1 4203.497,E2 4203.497} C_VEL
LIN {X 0,Y 534.698,Z 768.224,A -85,B 0,C 180,E1 4206.644,E2 4206.644} C_VEL
LIN {X 0,Y 533.074,Z 795.235,A -85,B 0,C 180,E1 4210.072,E2 4210.072} C_VEL
LIN {X 0,Y 531.951,Z 818.068,A -85,B 0,C 180,E1 4213.888,E2 4213.888} C_VEL
LIN {X 0,Y 531.351,Z 834.825,A -85,B 0,C 180,E1 4217.659,E2 4217.659} C_VEL
LIN {X 0,Y 531.168,Z 846.644,A -85,B 0,C 180,E1 4221.393,E2 4221.393} C_VEL
LIN {X 0,Y 531.007,Z 853.932,A -85,B 0,C 180,E1 4225.092,E2 4225.092} C_VEL
LIN {X 0,Y 530.985,Z 857.084,A -85,B 0,C 180,E1 4228.365,E2 4228.365} C_VEL
LIN {X 0,Y 531.072,Z 857.085,A -85,B 0,C 180,E1 4231.633,E2 4231.633} C_VEL
LIN {X 0,Y 531.107,Z 852.726,A -85,B 0,C 180,E1 4235.726,E2 4235.726} C_VEL
LIN {X 0,Y 531.223,Z 843.213,A -85,B 0,C 180,E1 4239.846,E2 4239.846} C_VEL
LIN {X 0,Y 531.668,Z 827.322,A -85,B 0,C 180,E1 4244.189,E2 4244.189} C_VEL
LIN {X 0,Y 532.553,Z 806.279,A -85,B 0,C 180,E1 4248.223,E2 4248.223} C_VEL
LIN {X 0,Y 533.991,Z 779.947,A -85,B 0,C 180,E1 4251.979,E2 4251.979} C_VEL
LIN {X 0,Y 535.825,Z 750.12,A -85,B 0,C 180,E1 4255.216,E2 4255.216} C_VEL
LIN {X 0,Y 537.833,Z 716.755,A -85,B 0,C 180,E1 4257.967,E2 4257.967} C_VEL
LIN {X 0,Y 539.959,Z 680.419,A -85,B 0,C 180,E1 4260.164,E2 4260.164} C_VEL
LIN {X 0,Y 541.615,Z 644.058,A -85,B 0,C 180,E1 4261.694,E2 4261.694} C_VEL
LIN {X 0,Y 542.668,Z 607.254,A -85,B 0,C 180,E1 4262.656,E2 4262.656} C_VEL
LIN {X 0,Y 542.14,Z 575.65,A -85,B 0,C 180,E1 4263.209,E2 4263.209} C_VEL
LIN {X 0,Y 530.262,Z 549.53,A -85,B 0,C 180,E1 4264.499,E2 4264.499} C_VEL
LIN {X 0,Y 530.289,Z 549.53,A -85,B 0,C 180,E1 4271.047,E2 4271.047} C_VEL
LIN {X 0,Y 530.256,Z 549.53,A -85,B 0,C 180,E1 4276.748,E2 4276.748} C_VEL
LIN {X 0,Y 530.206,Z 549.53,A -85,B 0,C 180,E1 4283.159,E2 4283.159} C_VEL
LIN {X 0,Y 530.377,Z 549.53,A -85,B 0,C 180,E1 4289.085,E2 4289.085} C_VEL
LIN {X 0,Y 530.379,Z 549.53,A -85,B 0,C 180,E1 4294.651,E2 4294.651} C_VEL
LIN {X 0,Y 530.489,Z 549.53,A -85,B 0,C 180,E1 4300.363,E2 4300.363} C_VEL
LIN {X 0,Y 530.626,Z 549.53,A -85,B 0,C 180,E1 4306.809,E2 4306.809} C_VEL
LIN {X 0,Y 530.715,Z 549.53,A -85,B 0,C 180,E1 4311.803,E2 4311.803} C_VEL
LIN {X 0,Y 530.852,Z 549.53,A -85,B 0,C 180,E1 4316.733,E2 4316.733} C_VEL
LIN {X 0,Y 530.963,Z 549.53,A -85,B 0,C 180,E1 4321.637,E2 4321.637} C_VEL
LIN {X 0,Y 530.844,Z 549.53,A -85,B 0,C 180,E1 4326.554,E2 4326.554} C_VEL
LIN {X 0,Y 530.642,Z 549.53,A -85,B 0,C 180,E1 4331.524,E2 4331.524} C_VEL
LIN {X 0,Y 530.554,Z 549.53,A -85,B 0,C 180,E1 4336.584,E2 4336.584} C_VEL
LIN {X 0,Y 530.507,Z 549.53,A -85,B 0,C 180,E1 4341.782,E2 4341.782} C_VEL
LIN {X 0,Y 530.331,Z 549.53,A -85,B 0,C 180,E1 4347.746,E2 4347.746} C_VEL
LIN {X 0,Y 530.255,Z 549.53,A -85,B 0,C 180,E1 4354.102,E2 4354.102} C_VEL
LIN {X 0,Y 530.228,Z 549.53,A -85,B 0,C 180,E1 4359.559,E2 4359.559} C_VEL
LIN {X 0,Y 530.222,Z 549.53,A -85,B 0,C 180,E1 4365.555,E2 4365.555} C_VEL
LIN {X 0,Y 530.173,Z 549.53,A -85,B 0,C 180,E1 4371.078,E2 4371.078} C_VEL
LIN {X 0,Y 530.351,Z 549.53,A -85,B 0,C 180,E1 4377.152,E2 4377.152} C_VEL
LIN {X 0,Y 530.293,Z 549.53,A -85,B 0,C 180,E1 4382.818,E2 4382.818} C_VEL
LIN {X 0,Y 530.428,Z 549.53,A -85,B 0,C 180,E1 4388.219,E2 4388.219} C_VEL
LIN {X 0,Y 530.537,Z 549.53,A -85,B 0,C 180,E1 4393.419,E2 4393.419} C_VEL
LIN {X 0,Y 530.61,Z 549.53,A -85,B 0,C 180,E1 4398.479,E2 4398.479} C_VEL
LIN {X 0,Y 530.703,Z 549.53,A -85,B 0,C 180,E1 4403.448,E2 4403.448} C_VEL
LIN {X 0,Y 530.768,Z 549.53,A -85,B 0,C 180,E1 4408.366,E2 4408.366} C_VEL
LIN {X 0,Y 530.742,Z 549.53,A -85,B 0,C 180,E1 4413.271,E2 4413.271} C_VEL
LIN {X 0,Y 530.638,Z 549.53,A -85,B 0,C 180,E1 4418.203,E2 4418.203} C_VEL
LIN {X 0,Y 530.541,Z 549.53,A -85,B 0,C 180,E1 4423.992,E2 4423.992} C_VEL
LIN {X 0,Y 530.524,Z 549.53,A -85,B 0,C 180,E1 4430.028,E2 4430.028} C_VEL
LIN {X 0,Y 530.512,Z 549.53,A -85,B 0,C 180,E1 4435.348,E2 4435.348} C_VEL
LIN {X 0,Y 530.283,Z 549.53,A -85,B 0,C 180,E1 4441.063,E2 4441.063} C_VEL
LIN {X 0,Y 530.278,Z 549.53,A -85,B 0,C 180,E1 4446.917,E2 4446.917} C_VEL
LIN {X 0,Y 530.308,Z 549.66,A -85,B 0,C 180,E1 4452.007,E2 4452.007} C_VEL
LIN {X 0,Y 540.878,Z 579.188,A -85,B 0,C 180,E1 4453.811,E2 4453.811} C_VEL
LIN {X 0,Y 538.967,Z 618.459,A -85,B 0,C 180,E1 4455.785,E2 4455.785} C_VEL
LIN {X 0,Y 536.777,Z 654.554,A -85,B 0,C 180,E1 4458.351,E2 4458.351} C_VEL
LIN {X 0,Y 534.778,Z 687.11,A -85,B 0,C 180,E1 4461.471,E2 4461.471} C_VEL
LIN {X 0,Y 533.183,Z 714.882,A -85,B 0,C 180,E1 4464.975,E2 4464.975} C_VEL
LIN {X 0,Y 532.07,Z 738.354,A -85,B 0,C 180,E1 4468.897,E2 4468.897} C_VEL
LIN {X 0,Y 531.463,Z 755.815,A -85,B 0,C 180,E1 4472.879,E2 4472.879} C_VEL
LIN {X 0,Y 531.109,Z 768.354,A -85,B 0,C 180,E1 4477.064,E2 4477.064} C_VEL
LIN {X 0,Y 530.961,Z 774.221,A -85,B 0,C 180,E1 4480.225,E2 4480.225} C_VEL
LIN {X 0,Y 530.909,Z 777.147,A -85,B 0,C 180,E1 4483.427,E2 4483.427} C_VEL
LIN {X 0,Y 530.967,Z 776.972,A -85,B 0,C 180,E1 4486.81,E2 4486.81} C_VEL
LIN {X 0,Y 531.064,Z 772.194,A -85,B 0,C 180,E1 4490.975,E2 4490.975} C_VEL
LIN {X 0,Y 531.314,Z 762.35,A -85,B 0,C 180,E1 4495.093,E2 4495.093} C_VEL
LIN {X 0,Y 531.715,Z 747.137,A -85,B 0,C 180,E1 4499.181,E2 4499.181} C_VEL
LIN {X 0,Y 532.555,Z 725.816,A -85,B 0,C 180,E1 4503.256,E2 4503.256} C_VEL
LIN {X 0,Y 534.047,Z 699.791,A -85,B 0,C 180,E1 4506.957,E2 4506.957} C_VEL
LIN {X 0,Y 535.9,Z 669.115,A -85,B 0,C 180,E1 4510.27,E2 4510.27} C_VEL
LIN {X 0,Y 538.07,Z 634.279,A -85,B 0,C 180,E1 4513.099,E2 4513.099} C_VEL
LIN {X 0,Y 540.121,Z 596.262,A -85,B 0,C 180,E1 4515.336,E2 4515.336} C_VEL
LIN {X 0,Y 540.543,Z 575.885,A -85,B 0,C 180,E1 4516.262,E2 4516.262} C_VEL
LIN {X 0,Y 532.957,Z 556.696,A -85,B 0,C 180,E1 4517.494,E2 4517.494} C_VEL
LIN {X 0,Y 528.477,Z 551.576,A -85,B 0,C 180,E1 4518.113,E2 4518.113} C_VEL
LIN {X 0,Y 522.873,Z 549.583,A -85,B 0,C 180,E1 4519.276,E2 4519.276} C_VEL
LIN {X 0,Y 522.511,Z 549.53,A -85,B 0,C 180,E1 4519.609,E2 4519.609} C_VEL
LIN {X 0,Y 522.552,Z 549.53,A -85,B 0,C 180,E1 4523.927,E2 4523.927} C_VEL
LIN {X 0,Y 522.36,Z 549.53,A -85,B 0,C 180,E1 4529.592,E2 4529.592} C_VEL
LIN {X 0,Y 522.308,Z 549.53,A -85,B 0,C 180,E1 4535.74,E2 4535.74} C_VEL
LIN {X 0,Y 522.392,Z 549.53,A -85,B 0,C 180,E1 4541.8,E2 4541.8} C_VEL
LIN {X 0,Y 522.283,Z 549.53,A -85,B 0,C 180,E1 4548.182,E2 4548.182} C_VEL
LIN {X 0,Y 522.398,Z 549.53,A -85,B 0,C 180,E1 4554.879,E2 4554.879} C_VEL
LIN {X 0,Y 536.071,Z 578.887,A -85,B 0,C 180,E1 4556.416,E2 4556.416} C_VEL
LIN {X 0,Y 535.423,Z 626.935,A -85,B 0,C 180,E1 4557.33,E2 4557.33} C_VEL
LIN {X 0,Y 533.84,Z 665.186,A -85,B 0,C 180,E1 4558.674,E2 4558.674} C_VEL
LIN {X 0,Y 531.691,Z 702.644,A -85,B 0,C 180,E1 4560.673,E2 4560.673} C_VEL
LIN {X 0,Y 529.33,Z 737.098,A -85,B 0,C 180,E1 4563.223,E2 4563.223} C_VEL
LIN {X 0,Y 527.222,Z 768.224,A -85,B 0,C 180,E1 4566.293,E2 4566.293} C_VEL
LIN {X 0,Y 525.422,Z 795.234,A -85,B 0,C 180,E1 4569.769,E2 4569.769} C_VEL
LIN {X 0,Y 524.21,Z 818.066,A -85,B 0,C 180,E1 4573.643,E2 4573.643} C_VEL
LIN {X 0,Y 523.529,Z 834.826,A -85,B 0,C 180,E1 4577.472,E2 4577.472} C_VEL
LIN {X 0,Y 523.251,Z 847.612,A -85,B 0,C 180,E1 4581.681,E2 4581.681} C_VEL
LIN {X 0,Y 523.108,Z 853.932,A -85,B 0,C 180,E1 4585.018,E2 4585.018} C_VEL
LIN {X 0,Y 523.101,Z 857.084,A -85,B 0,C 180,E1 4588.341,E2 4588.341} C_VEL
LIN {X 0,Y 523.182,Z 857.085,A -85,B 0,C 180,E1 4591.658,E2 4591.658} C_VEL
LIN {X 0,Y 523.216,Z 852.726,A -85,B 0,C 180,E1 4595.812,E2 4595.812} C_VEL
LIN {X 0,Y 523.34,Z 843.214,A -85,B 0,C 180,E1 4599.996,E2 4599.996} C_VEL
LIN {X 0,Y 523.827,Z 827.815,A -85,B 0,C 180,E1 4604.288,E2 4604.288} C_VEL
LIN {X 0,Y 524.848,Z 806.277,A -85,B 0,C 180,E1 4608.5,E2 4608.5} C_VEL
LIN {X 0,Y 526.399,Z 780.334,A -85,B 0,C 180,E1 4612.263,E2 4612.263} C_VEL
LIN {X 0,Y 528.458,Z 750.389,A -85,B 0,C 180,E1 4615.566,E2 4615.566} C_VEL
LIN {X 0,Y 530.703,Z 717.26,A -85,B 0,C 180,E1 4618.338,E2 4618.338} C_VEL
LIN {X 0,Y 532.974,Z 681.559,A -85,B 0,C 180,E1 4620.539,E2 4620.539} C_VEL
LIN {X 0,Y 534.802,Z 645.738,A -85,B 0,C 180,E1 4622.085,E2 4622.085} C_VEL
LIN {X 0,Y 536.029,Z 607.254,A -85,B 0,C 180,E1 4623.112,E2 4623.112} C_VEL
LIN {X 0,Y 535.55,Z 578.326,A -85,B 0,C 180,E1 4623.63,E2 4623.63} C_VEL
LIN {X 0,Y 522.338,Z 549.53,A -85,B 0,C 180,E1 4625.123,E2 4625.123} C_VEL
LIN {X 0,Y 522.412,Z 549.53,A -85,B 0,C 180,E1 4631.109,E2 4631.109} C_VEL
LIN {X 0,Y 522.334,Z 549.53,A -85,B 0,C 180,E1 4636.44,E2 4636.44} C_VEL
LIN {X 0,Y 522.247,Z 549.53,A -85,B 0,C 180,E1 4642.501,E2 4642.501} C_VEL
LIN {X 0,Y 522.431,Z 549.53,A -85,B 0,C 180,E1 4648.561,E2 4648.561} C_VEL
LIN {X 0,Y 522.421,Z 549.53,A -85,B 0,C 180,E1 4654.237,E2 4654.237} C_VEL
LIN {X 0,Y 522.498,Z 549.53,A -85,B 0,C 180,E1 4659.656,E2 4659.656} C_VEL
LIN {X 0,Y 522.642,Z 549.53,A -85,B 0,C 180,E1 4664.891,E2 4664.891} C_VEL
LIN {X 0,Y 522.774,Z 549.53,A -85,B 0,C 180,E1 4669.997,E2 4669.997} C_VEL
LIN {X 0,Y 522.957,Z 549.53,A -85,B 0,C 180,E1 4676.684,E2 4676.684} C_VEL
LIN {X 0,Y 523.055,Z 549.53,A -85,B 0,C 180,E1 4681.662,E2 4681.662} C_VEL
LIN {X 0,Y 522.915,Z 549.53,A -85,B 0,C 180,E1 4686.654,E2 4686.654} C_VEL
LIN {X 0,Y 522.711,Z 549.53,A -85,B 0,C 180,E1 4691.702,E2 4691.702} C_VEL
LIN {X 0,Y 522.593,Z 549.53,A -85,B 0,C 180,E1 4697.046,E2 4697.046} C_VEL
LIN {X 0,Y 522.565,Z 549.53,A -85,B 0,C 180,E1 4702.13,E2 4702.13} C_VEL
LIN {X 0,Y 522.435,Z 549.53,A -85,B 0,C 180,E1 4707.629,E2 4707.629} C_VEL
LIN {X 0,Y 522.338,Z 549.53,A -85,B 0,C 180,E1 4713.421,E2 4713.421} C_VEL
LIN {X 0,Y 522.329,Z 549.53,A -85,B 0,C 180,E1 4719.624,E2 4719.624} C_VEL
LIN {X 0,Y 522.359,Z 549.53,A -85,B 0,C 180,E1 4724.082,E2 4724.082} C_VEL
LIN {X 0,Y 522.261,Z 549.53,A -85,B 0,C 180,E1 4730.374,E2 4730.374} C_VEL
LIN {X 0,Y 522.434,Z 549.53,A -85,B 0,C 180,E1 4736.59,E2 4736.59} C_VEL
LIN {X 0,Y 522.386,Z 549.53,A -85,B 0,C 180,E1 4742.372,E2 4742.372} C_VEL
LIN {X 0,Y 522.513,Z 549.53,A -85,B 0,C 180,E1 4748.016,E2 4748.016} C_VEL
LIN {X 0,Y 522.607,Z 549.53,A -85,B 0,C 180,E1 4753.16,E2 4753.16} C_VEL
LIN {X 0,Y 522.698,Z 549.53,A -85,B 0,C 180,E1 4758.302,E2 4758.302} C_VEL
LIN {X 0,Y 522.792,Z 549.53,A -85,B 0,C 180,E1 4763.348,E2 4763.348} C_VEL
LIN {X 0,Y 522.875,Z 549.53,A -85,B 0,C 180,E1 4768.341,E2 4768.341} C_VEL
LIN {X 0,Y 522.837,Z 549.53,A -85,B 0,C 180,E1 4773.321,E2 4773.321} C_VEL
LIN {X 0,Y 522.725,Z 549.53,A -85,B 0,C 180,E1 4778.328,E2 4778.328} C_VEL
LIN {X 0,Y 522.668,Z 549.53,A -85,B 0,C 180,E1 4783.401,E2 4783.401} C_VEL
LIN {X 0,Y 522.606,Z 549.53,A -85,B 0,C 180,E1 4788.584,E2 4788.584} C_VEL
